	    #sR_TRIG_FlowSplitterDownTime(CLK := #sx_AutomaticActive AND NOT #sx_Ready);     // Rising edge conveyor conveyor down

	    #sR_TRIG_AirPressureError(CLK := NOT #ix_AirPressureOk);                         // Rising edge air pressure error

	    #sR_TRIG_DebrisDetected(CLK := #ix_DebrisSensor);                                // Rising edge debris detection

	    #sR_TRIG_EnconderError(CLK := #ix_FlowSplitterEncoderError);                    // Rising edge encoder error

	    #sR_TRIG_Mode1(CLK := (#si_Mode = 1));                                          // Rising edge Mode 1

	    #sR_TRIG_Mode2(CLK := (#si_Mode = 2));                                          // Rising edge Mode 2

	    #sR_TRIG_Mode3(CLK := (#si_Mode = 3));                                          // Rising edge Mode 3

	    #sR_TRIG_Mode4(CLK := (#si_Mode = 4));                                          // Rising edge Mode 4

	    #sR_TRIG_Mode5(CLK := (#si_Mode = 5));                                          // Rising edge Mode 5

	    #sR_TRIG_EnergySave(CLK := #sUDT_CommonStatus.EnergySave);                     // Rising edge trigger Energy save mode.

	    // Timers

	    #PEC_TimerOnOffDelay(iudi_OnDelayTime := #iUDT_FlowSplitterConfiguration.PEC_EoSTimeOnDelay,                       // Off delay time to filter PEC signal
	                         iudi_OffDelayTime := #iUDT_FlowSplitterConfiguration.PEC_EoSTimeOffDelay,                     // On delay time to filter PEC signal
	                         ix_SignalToDelay := #ix_PECEos,                                                               // PEC input signal
	                         ix_Enable := #iUDT_FlowSplitterConfiguration.PEC_Present,                                     // PEC present bit is true if the flow splitter is equiped with PEC
	                         qx_DelayedSignal => #sx_PEC_EoSFiltered);                                                      // PEC signal filtered

	    #PEC_ChuteTimerOnOffDelay(iudi_OnDelayTime := #iUDT_FlowSplitterConfiguration.PEC_FilterChuteTimeOnDelay,          // Off delay time to filter chute PEC signal
	                              iudi_OffDelayTime := #iUDT_FlowSplitterConfiguration.PEC_FilterChuteTimeOffDelay,        // On delay time to filter chute PEC signal
	                              ix_SignalToDelay := #ix_PECDivertChute,                                                  // PEC chute signal
	                              ix_Enable := TRUE,                                                                        // Enable function
	                              qx_DelayedSignal => #sx_PEC_ChuteFiltered);                                               // PEC chute siganl filtered

	    #PEC_UpstreamTimerOnOffDelay(iudi_OnDelayTime := #iUDT_FlowSplitterConfiguration.PEC_FilterUpstreamTimeOnDelay,    // On delay time to filter upstream PEC
	                                 iudi_OffDelayTime := #iUDT_FlowSplitterConfiguration.PEC_FilterUpstreamTimeOffDelay,  // Off delay time to filter upstream PEC
	                                 ix_SignalToDelay := #ix_PECUpstream,                                                  // Signal to filter upstream PEC
	                                 ix_Enable := TRUE,                                                                     // Function enable
	                                 qx_DelayedSignal => #sx_PEC_UpstreamFiltered);                                         // Upstream PEC signal filtered

	    #sFB_DivertsActivationTimer(iudi_OnDelayTime := 0,
	                                iudi_OffDelayTime := #iUDT_FlowSplitterConfiguration.DivertsTimeActivation,                // Off delay to pop-up diverts
	                                ix_SignalToDelay := NOT #sx_PEC_UpstreamFiltered,                                           // Upstream signal filtered,
	                                ix_Enable := TRUE,
	                                qx_DelayedSignal => #sx_EnableDiverts);                                                     // Enabling diverts pop-up

	END_REGION

	REGION 2 - Reset faults

	    // Send reset request TO interface UDT
	    #iqUDT_FlowSplitterInterface.InternalErrorReset := #iqUDT_EquipmentControl.Command.Reset;
	    #iqUDT_FlowSplitterInterface.ResetStatistics := #iqUDT_EquipmentControl.Command.ResetData;

	    // Reset errors
	    // Reset PEC Jam if PEC is clear and reset command is received.
	    IF #iqUDT_EquipmentControl.Command.Reset THEN                      // Reset bit from control block

	        IF #ix_PECEos = TRUE THEN
	            #sUDT_HMIStatus.Specific.PEC_EoSJam := FALSE;                     // PEC jam reset
	        END_IF;

	        IF #ix_DebrisSensor = TRUE THEN
	            #sUDT_HMIStatus.Specific.Debris := FALSE;                         // Debris fault reset
	        END_IF;

	        IF #ix_PECDivertChute = TRUE THEN
	            #sUDT_HMIStatus.Specific.PEC_DivertChuteJam := FALSE;             // Divert chute jam reset
	        END_IF;

	        IF #ix_AirPressureOk = TRUE THEN
	            #sUDT_HMIStatus.Specific.AirPressure := FALSE;                    // Air pressure error reset
	        END_IF;

	        IF #ix_FlowSplitterEncoderError = FALSE THEN
	            #sUDT_HMIStatus.Specific.EncoderError := FALSE;                   // Encoder error reset
	        END_IF;

	    END_IF;

	    // Error
	    #sUDT_CommonStatus.Error := NOT #ix_SafetyOk                               // safety error status
	    OR #sUDT_HMIStatus.Specific.EncoderError                                   // Enconder error status
	    OR #sUDT_HMIStatus.Specific.PEC_EoSJam                                     // PEC blockage error status
	    OR #sUDT_HMIStatus.Specific.PEC_DivertChuteJam                             // PEC divert chute blockage error status
	    OR #sUDT_HMIStatus.Specific.Debris                                         // Debris detected error status
	    OR #sUDT_HMIStatus.Specific.DivertsActivationError                         // Diverts position error status
	    OR #iqUDT_FlowSplitterInterface.InternalErrorVFD                           // Internal VFD error status
	    OR NOT #ix_Connected                                                        // Isolator switch error status
	    OR #iqUDT_FlowSplitterInterface.InternalErrorPEC;                          // External PEC fault
	    // Warning
	    #sUDT_CommonStatus.Warning := #sUDT_HMIStatus.Specific.AirPressure;       // Air pressure status;

	    // Ready
	    #sx_Ready := NOT #sUDT_CommonStatus.Error                                  // Ready bit is set true when common error status its false
	    AND #ix_24vOk                                                               // 24V is okay
	    AND #ix_400vOk                                                              // 400V is okay
	    AND NOT #iqUDT_FlowSplitterInterface.ConfigurationError;                   // not configuration error

	END_REGION

	REGION 3 - Stop conveyor

	    // Conditions to stop conveyor
	    IF ((#sF_TRIG_RunManual.Q OR #sF_TRIG_Jog.Q) AND #sx_ManualModeActive)                        // If in manula mode and Rising or falling edge for jog occur
	        OR (NOT #iqUDT_EquipmentControl.Command.AutomaticOn AND NOT #sx_ManualModeActive)      // or Not automatic ON and Not in manual mode
	        OR (NOT #sx_Ready AND NOT #sx_ManualModeActive)                                         // Or not ready and not in automatic mode
	        OR (#sR_TRIG_ManualMode.Q OR #sF_TRIG_ManualMode.Q)                                       // or Rising edge or falling edge of manual mode active command occur
	        OR NOT #ix_SafetyOk                                                                     // or safety not ok

	    THEN
	        //  Order to stop VFD
	        #iqUDT_FlowSplitterInterface.RunFwd := FALSE;                  // Reset order to VFD run in forward direction
	        #iqUDT_FlowSplitterInterface.RunRvs := FALSE;                  // Reset order to VFD run in reverse direction
	        #iqUDT_HandShakeUp.RTR := FALSE;                               // Reset the bit ready to receive
	        #iqUDT_HandShakeUp.CascadeStartUp := FALSE;                    // Reset cascade start up bit

	        #sx_AutomaticActive := FALSE;                                   // Automatic mode is disable
	        #sx_StartReceived := FALSE;                                     // Clear start receive bit

	        #sx_Zone1_Divert := FALSE;                                      // Reset diverts from zone 1
	        #sx_Zone2_Divert := FALSE;                                      // Reset diverts from zone 2

	        #sx_Switch1To3 := FALSE;                                        // Reset switch from mode 1 to mode 3 auxiliary bit
	        #sx_Switch3To1 := FALSE;                                        // Reset switch from mode 3 to mode 1 auxiliary bit
	    END_IF;

	END_REGION

	REGION 4 - Start
	    // Save Start bit request
	    IF NOT #sx_ManualModeActive                                         // If Manual mode iis not active
	        AND #sx_Ready                                                   // and Flow splitter is ready
	        AND #iqUDT_EquipmentControl.Command.Start                      // Start command from control block received
	        AND #iqUDT_EquipmentControl.Command.AutomaticOn                // Automatic on signal from control block is active
	    THEN                                                                // then
	        #sx_StartReceived := TRUE;                                      // Set start received bit
	    END_IF;

	    // Cascade mode

	    CASE #si_Mode OF
	        1:  // Statement section case 1 (Flow splitter in straight direction)
	            IF #sx_StartReceived                                                 // If Start received memory bit is active
	                AND (#iqUDT_HandShakeStraight.CascadeStartUp                    // And Cascade start bit from downstream straight conveyor handshake is active
	                OR #iUDT_FlowSplitterConfiguration.FirstConveyorToStart)        // Or flow splitter conveyor is the first conveyor to start
	            THEN                                                                 // then
	                #sx_AutomaticActive := TRUE;                                     // Automatic active is set true
	                #sx_StartReceived := FALSE;                                      // and reset start received memory bit
	            END_IF;
	            ;
	        3:  // Statement section case 3 (Flow splitter in divert direction)
	            IF #sx_StartReceived                                                 // If Start received memory bit is active
	                AND (#iqUDT_HandShakeDivert.CascadeStartUp                      // And Cascade start bit from downstream divert conveyor handshake is avtive
	                OR #iUDT_FlowSplitterConfiguration.FirstConveyorToStart)        // Or flow splitter conveyor is the first conveyor to start
	            THEN                                                                 // Then
	                #sx_AutomaticActive := TRUE;                                     //  Automatic active is set true
	                #sx_StartReceived := FALSE;                                      //and reset start received memory bit
	            END_IF;
	            ;
	        ELSE  // Statement section ELSE
	            IF #sx_StartReceived                                                 // If Start received memory bit is activ
	                AND (#iqUDT_HandShakeStraight.CascadeStartUp                    // And Cascade start bit from downstream straight conveyor handshake is active
	                AND #iqUDT_HandShakeDivert.CascadeStartUp                       // And Cascade start bit from downstream divert conveyor handshake is active
	                OR #iUDT_FlowSplitterConfiguration.FirstConveyorToStart)        // Or flow splitter conveyor is the first conveyor to start
	            THEN                                                                 // Then
	                #sx_AutomaticActive := TRUE;                                     // Automatic active is set true
	                #sx_StartReceived := FALSE;                                      // and reset start received memory bit
	            END_IF;
	            ;
	    END_CASE;

	    //Timer to cascade mode

	    #sFB_CascadeModeTimer(iudi_OnDelayTime := #iUDT_FlowSplitterConfiguration.CascadeTimeOnDelay,      // Cascade mode timer
	                          ix_SignalToDelay := #sx_AutomaticActive,                                      // Signal to activate the timer
	                          ix_Enable := #sx_Ready,                                                       // Bit ready to enable cascade mode
	                          qx_DelayedSignal => #iqUDT_HandShakeUp.CascadeStartUp);                      // Cascade mode signal to upstream

	END_REGION

	REGION 5 - Manual mode

	    // Manual mode activation
	    #sx_ManualModeActive := #iqUDT_FlowSplitterCommand.ManualMode                                  // Manual mode is active if the bits that activate manual mode is active from hmi or from control block
	    OR #iqUDT_EquipmentControl.Command.ManualMode;

	    //Send manual mode active to PEC/VFD blocks to supress errors
	    #iqUDT_FlowSplitterInterface.ManualModeActive := #sx_ManualModeActive;

	    //When the system is not any more in manual mode or when fatal error occurs the HMI commands should be reset

	    IF NOT #ix_SafetyOk
	        OR NOT #ix_24vOk                                                        // 24V error status
	        OR NOT #ix_400vOk                                                       // 400V error status
	        OR NOT #ix_HardwareOk                                                   // Profinet error status
	        OR #iqUDT_FlowSplitterInterface.ConfigurationError                          // No configuration err
	        OR #iqUDT_FlowSplitterInterface.InternalErrorVFD
	        OR #iqUDT_FlowSplitterInterface.Disconnected
	        OR NOT #sx_ManualModeActive
	    THEN
	        #iqUDT_FlowSplitterCommand.ManualStartStop := FALSE;
	        #iqUDT_FlowSplitterCommand.ManualFullSpeed := FALSE;
	        #iqUDT_FlowSplitterCommand.ManualJog := FALSE;
	    END_IF;

	    // Manual mode force disable
	    IF #iqUDT_EquipmentControl.Command.DisableManualMode THEN
	        #iqUDT_FlowSplitterCommand.ManualMode := False;
	        #iqUDT_FlowSplitterCommand.ManualFullSpeed := False;
	        #iqUDT_FlowSplitterCommand.ManualJog := False;
	        #iqUDT_FlowSplitterCommand.ManualStartStop := False;
	    END_IF;

	    // Start/Stop in manual mode
	    IF #sx_ManualModeActive THEN                                            // If Manual mode is active then check prestart status for manual mode
	        #sx_PreStartManual := #ix_SafetyOk                                  // If Safety is Okay
	        AND #ix_Connected                                                   // And Isolator switch is connected
	        AND #ix_HardwareOk                                                  // And Profinet connection is okay
	        AND NOT #iqUDT_FlowSplitterInterface.InternalErrorVFD;             // Add no error on VFD // Then conveyor is allowed to run in manual mode.

	        IF (#sx_PreStartManual                                                              // If Pre start conditions to run in manual mode is okay
	            AND (#sR_TRIG_RunManual.Q AND NOT #iqUDT_FlowSplitterCommand.ManualJog)         // and rising edge to run in manual mode is detected and it is not running in jogging mode
	            OR (#sR_TRIG_Jog.Q AND NOT #iqUDT_FlowSplitterCommand.ManualStartStop))         // Or rising edge to start jogging is detected and it is not running in manual mode
	        THEN
	            #iqUDT_EquipmentControl.Request.SignalingRequest := TRUE;                      //then Request signaling to control block before conveyor run in manual mode
	        END_IF;

	        // To Run conveyor forward in manual mode
	        #iqUDT_FlowSplitterInterface.RunFwd := #sx_PreStartManual          // Prestart conditions to run in manual mode is active
	        AND NOT #iqUDT_EquipmentControl.Request.SignalingRequest           // And Signaling request done
	        AND (#iqUDT_FlowSplitterCommand.ManualStartStop                    // And Command to manual Run or manual jog is active
	        OR #iqUDT_FlowSplitterCommand.ManualJog);                          // Then run motor in forward direction

	        // Flow splitter belt should not run in reverse direction
	        #iqUDT_FlowSplitterInterface.RunRvs := FALSE;

	        // Pop up diverts in manual mode
	        #sx_Zone1_Divert := #sx_PreStartManual AND #iqUDT_FlowSplitterCommand.Zone1DivertActivation;          // Output bit to active zone 1 diverts
	        #sx_Zone2_Divert := #sx_PreStartManual AND #iqUDT_FlowSplitterCommand.Zone2DivertActivation;          // Output bit to active zone 2 diverts

	    END_IF;

	END_REGION

	REGION 6 - Automatic mode active

	    IF NOT #sx_ManualModeActive THEN                                        // Manual mode is not active
	        IF #sx_AutomaticActive AND #sx_Ready THEN                           // Automatic mode active AND ready

	            #iqUDT_HandShakeUp.RTR := #iqUDT_FlowSplitterInterface.VFDatSpeed;            // Ready to receive handshake to upstream if VFD is at speed

	            CASE #si_Mode OF                                                // Operation mode case selection

	                1:  // 100% straight

	                    // Order to VFD to run
	                    #iqUDT_FlowSplitterInterface.RunFwd := NOT #ix_ExternalRequestHold             // Halt request is not active
	                    AND #iqUDT_HandShakeStraight.RTR                                               // Ready to receive active
	                    AND NOT #sx_EnergySaveActive;                                                   // Energy save is not active

	                    #sx_Zone2_Divert := FALSE;                                                      // Output bit to active zone 2 diverts
	                    #sx_Zone1_Divert := #sx_Switch3To1;                                             // Output bit to active zone 1 diverts

	                    IF #sx_Switch3To1 THEN                                                          // Memory bit switch from mode 3 to mode 1
	                        IF "DB_Memory".OS_1sec THEN                                                 // Memory bit 1 second trigger
	                            #si_SwitchDelay += 1;                                                   // Memory integer to count time to delay switch
	                        END_IF;

	                        IF #si_SwitchDelay >= #iUDT_FlowSplitterConfiguration.DivertSwitchDelay THEN    // Comparation between memory integer switch delay and configuration divert switch delay
	                            #si_SwitchDelay := 0;                                                   // Reset memory integer switch delay counter
	                            #sx_Switch3To1 := FALSE;                                                // Reset switch from mode 3 to mode 1 memory bit
	                        END_IF;
	                    END_IF;

	                    #sx_Switch1To3 := TRUE;                                                         // Set memory bit switch from mode 1 to mode 3
	                    ;

	                2:  // 50% straight - 50% divert

	                    #iqUDT_FlowSplitterInterface.RunFwd := ((#iqUDT_HandShakeStraight.RTR         // Ready to receive downstream straight
	                    AND #iqUDT_HandShakeDivert.RTR)                                                // Ready to receive downstream divert chute
	                    OR (#iUDT_FlowSplitterConfiguration.OnFlyChangeOfMode                          // On fly change mode
	                    AND (#iqUDT_HandShakeStraight.RTR                                              // Ready to receive downstream straight
	                    OR (#iqUDT_HandShakeDivert.RTR AND NOT #sUDT_HMIStatus.Specific.AirPressure))))// Ready to receive downstream divert chute
	                    //   AND (NOT #i_UDT_FlowSplitterConfiguration.OnFlyChangeOfMode
	                    //   AND NOT #s_UDT_HMIStatus.Specific.AirPressure)
	                    AND NOT #ix_ExternalRequestHold                                                // External requesto to halt
	                    AND NOT #sx_EnergySaveActive;                                                   // Energy save is not active

	                    #sx_Zone1_Divert := (#iqUDT_HandShakeDivert.RTR                                // Ready to receive downstream divert chute
	                    OR NOT #iqUDT_HandShakeStraight.RTR                                            // Ready to receive downstream straight
	                    OR NOT #iUDT_FlowSplitterConfiguration.OnFlyChangeOfMode)                      // On fly change mode
	                    AND NOT #sUDT_HMIStatus.Specific.AirPressure;                                         // And Air pressure is OK

	                    #sx_Zone2_Divert := (#iUDT_FlowSplitterConfiguration.OnFlyChangeOfMode         // On fly change mode
	                    AND NOT #iqUDT_HandShakeStraight.RTR                                           // Ready to receive downstream straight
	                    AND #iqUDT_HandShakeDivert.RTR)
	                    AND NOT #sUDT_HMIStatus.Specific.AirPressure;                                         // Ready to receive downstream divert chute

	                    #sx_Switch1To3 := FALSE;                                                        // Switch from mode 1 to mode 3
	                    #sx_Switch3To1 := FALSE;                                                        // Switch from mode 3 to mode 1
	                    ;

	                3:  // 0% straight - 100% divert

	                    // Order to VFD to run
	                    #iqUDT_FlowSplitterInterface.RunFwd := NOT #ix_ExternalRequestHold             // Halt request is not active
	                    AND #iqUDT_HandShakeDivert.RTR                                                 // Handshake Ready to receive from downstream divert conveyor
	                    AND NOT #sUDT_HMIStatus.Specific.AirPressure
	                    AND NOT #sx_EnergySaveActive;                                                   // Energy save is not active

	                    #sx_Zone1_Divert := NOT #sUDT_HMIStatus.Specific.AirPressure;                         // Output bit to active zone 1 diverts
	                    #sx_Zone2_Divert := NOT #sx_Switch1To3 AND NOT #sUDT_HMIStatus.Specific.AirPressure;  // Output bit to active zone 2 diverts

	                    IF #sx_Switch1To3 THEN                                                          // Memory bit switch mode 1 to mode 3
	                        IF "DB_Memory".OS_1sec THEN                                                 // Memory bit 1 second trigger
	                            #si_SwitchDelay += 1;                                                   // Memory integer to count time to delay switch
	                        END_IF;

	                        IF #si_SwitchDelay > #iUDT_FlowSplitterConfiguration.DivertSwitchDelay     // Comparation between memory integer switch delay and configuration divert switch delay
	                        THEN
	                            #si_SwitchDelay := 0;                                                   // Reset memory integer switch delay counter
	                            #sx_Switch1To3 := FALSE;                                                // Reset switch from mode 1 to mode 3 memory bit
	                        END_IF;
	                    END_IF;
	                    #sx_Switch3To1 := TRUE;                                                         // Set memory bit switch from mode 3 to mode 1
	                    ;

	                4:  // Based on time

	                    #iqUDT_FlowSplitterInterface.RunFwd := ((#iqUDT_HandShakeStraight.RTR         // Ready to receive downstream straight
	                    AND #iqUDT_HandShakeDivert.RTR)                                                // Ready to receive downstream divert chute
	                    OR (#iUDT_FlowSplitterConfiguration.OnFlyChangeOfMode                          // On fly change mode
	                    AND (#iqUDT_HandShakeStraight.RTR                                              // Ready to receive downstream straight
	                    OR (#iqUDT_HandShakeDivert.RTR AND NOT #sUDT_HMIStatus.Specific.AirPressure))))      // Ready to receive downstream divert chute
	                    //  AND (NOT #i_UDT_FlowSplitterConfiguration.OnFlyChangeOfMode
	                    //  AND NOT #s_UDT_HMIStatus.Specific.AirPressure)
	                    AND NOT #ix_ExternalRequestHold                                                 // External requesto to halt
	                    AND NOT #sx_EnergySaveActive;                                                   // Energy save is not active

	                    #sx_Switch1To3 := FALSE;                                                        // Reset switch from mode 1 to mode 3 memory bit
	                    #sx_Switch3To1 := FALSE;                                                        // Reset switch from mode 3 to mode 1 memory bit

	                    #si_Mode4DivertTime := REAL_TO_INT(#iqUDT_FlowSplitterCommand.PercentageSplit * #iUDT_FlowSplitterConfiguration.TimeBasedSplit) / 100;      // Memory integer to calculate time base

	                    IF "DB_Memory".OS_1sec AND #iqUDT_HandShakeDivert.RTR THEN                     // Memory bit 1 second trigger and Handshake bit ready to receive to upstream
	                        #si_Mode4AuxTimer += 1;                                                     // Increment counter to time base mode
	                    END_IF;

	                    #tx_AuxBaseTimeDivert1 := FALSE;                                                // Auxiliary base time divert zone 1
	                    #tx_AuxBaseTimeDivert2 := FALSE;                                                // Auxiliary base time divert zone 2

	                    IF (#si_Mode4AuxTimer <= #si_Mode4DivertTime)                                   // If the counter time is lower than calculated time from configuration
	                    THEN
	                        #tx_AuxBaseTimeDivert1 := TRUE;                                             // Auxiliary base time divert zone 1
	                        #tx_AuxBaseTimeDivert2 := TRUE;                                             // Auxiliary base time divert zone 2
	                    END_IF;

	                    IF (#si_Mode4AuxTimer > #si_Mode4DivertTime)                                    // If the counter time is bigger than calculated time from configuration
	                        AND (#si_Mode4AuxTimer < #iUDT_FlowSplitterConfiguration.TimeBasedSplit)   // If the counter time is lower than time based split configured
	                    THEN
	                        #tx_AuxBaseTimeDivert1 := FALSE;                                            // Auxiliary base time divert zone 1
	                        #tx_AuxBaseTimeDivert2 := FALSE;                                            // Auxiliary base time divert zone 2
	                    END_IF;

	                    IF (#si_Mode4AuxTimer >= #iUDT_FlowSplitterConfiguration.TimeBasedSplit) THEN  // If the counter time is bigger or equal than time based split configured
	                        #si_Mode4AuxTimer := 0;                                                     // Reset counter time
	                    END_IF;

	                    IF (#iqUDT_HandShakeDivert.RTR                                                 // Ready to receive downstream divert chute
	                        AND ((#tx_AuxBaseTimeDivert1 AND #tx_AuxBaseTimeDivert2)
	                        OR (NOT #iqUDT_HandShakeStraight.RTR AND #iUDT_FlowSplitterConfiguration.OnFlyChangeOfMode)))
	                        AND NOT #sUDT_HMIStatus.Specific.AirPressure
	                    THEN
	                        #sx_Zone1_Divert := TRUE;
	                        #sx_Zone2_Divert := TRUE;

	                    ELSIF #iqUDT_HandShakeStraight.RTR
	                        AND ((NOT #tx_AuxBaseTimeDivert1 AND NOT #tx_AuxBaseTimeDivert2)
	                        OR (NOT #iqUDT_HandShakeDivert.RTR AND #iUDT_FlowSplitterConfiguration.OnFlyChangeOfMode))
	                        OR #sUDT_HMIStatus.Specific.AirPressure
	                    THEN
	                        #sx_Zone1_Divert := FALSE;
	                        #sx_Zone2_Divert := FALSE;
	                    END_IF
	                    ;

	                5:  // Semi automatic mode

	                    #iqUDT_FlowSplitterInterface.RunFwd := NOT #ix_ExternalRequestHold     // External requesto to halt
	                    AND NOT #sx_EnergySaveActive                                            // Energy save is not active
	                    AND ((#iqUDT_HandShakeStraight.RTR                                     // Ready to receive downstream straight
	                    AND NOT #iqUDT_FlowSplitterCommand.Zone1DivertActivation               // Command divert activation zone 1
	                    AND NOT #iqUDT_FlowSplitterCommand.Zone2DivertActivation)              // Command divert activation zone 2
	                    OR (#iqUDT_HandShakeDivert.RTR                                         // Ready to receive downstream divert chute
	                    AND #iqUDT_FlowSplitterCommand.Zone1DivertActivation                   // Command divert activation zone 1
	                    AND #iqUDT_FlowSplitterCommand.Zone2DivertActivation                   // Command divert activation zone 2
	                    AND NOT #sUDT_HMIStatus.Specific.AirPressure)                                 // Air preassure is OK
	                    OR (#iqUDT_HandShakeStraight.RTR                                       // Ready to receive downstream straight
	                    AND #iqUDT_HandShakeDivert.RTR                                         // Ready to receive downstream divert chute
	                    AND #iqUDT_FlowSplitterCommand.Zone1DivertActivation                   // Command divert activation zone 1
	                    AND NOT #iqUDT_FlowSplitterCommand.Zone2DivertActivation               // Command divert activation zone 2
	                    AND NOT #sUDT_HMIStatus.Specific.AirPressure));

	                    #sx_Zone1_Divert := #iqUDT_FlowSplitterCommand.Zone1DivertActivation   // Command divert activation zone 1
	                    AND NOT #sUDT_HMIStatus.Specific.AirPressure;

	                    #sx_Zone2_Divert := #iqUDT_FlowSplitterCommand.Zone2DivertActivation   // Command divert activation zone 2
	                    AND NOT #sUDT_HMIStatus.Specific.AirPressure;

	                    #sx_Switch1To3 := FALSE;                                                // Reset switch from mode 1 to mode 3 memory bit
	                    #sx_Switch3To1 := FALSE;                                                // Reset switch from mode 3 to mode 1 memory bit
	                    ;
	            END_CASE;

	            // Flow splitter end OF section PEC jam

	            IF #iUDT_FlowSplitterConfiguration.PEC_Present THEN

	                IF NOT #sx_PEC_EoSFiltered AND #ix_HardwareOk THEN                                      // Photo eye blocked
	                    #si_AuxJamDisplacement += #iqUDT_FlowSplitterInterface.Displacement;               // Increases displacement values in auxiliary variable
	                ELSE
	                    #si_AuxJamDisplacement := 0;                                                        // Reset jam auxiliary counter variable
	                END_IF;

	                IF #si_AuxJamDisplacement > #iUDT_FlowSplitterConfiguration.JamDisplacementLimit THEN  // Compare jam auxiliary counter with displacement jam configured
	                    #sUDT_HMIStatus.Specific.PEC_EoSJam := TRUE;                                              // PEC jam status set true
	                END_IF;

	            END_IF;

	            // Chute PEC jam

	            IF #iUDT_FlowSplitterConfiguration.PEC_ChutePesent THEN
	                IF NOT #sx_PEC_ChuteFiltered AND #ix_HardwareOk THEN
	                    #si_AuxJamDivertChuteDisplacement += #iqUDT_FlowSplitterInterface.Displacement;
	                ELSE
	                    #si_AuxJamDivertChuteDisplacement := 0;
	                END_IF;

	                IF #si_AuxJamDivertChuteDisplacement > #iUDT_FlowSplitterConfiguration.DivertChuteJamDisplacLimit THEN     // Compare jam auxiliary counter with displacement jam configured
	                    #sUDT_HMIStatus.Specific.PEC_DivertChuteJam := TRUE;                                                          // PEC jam status set true
	                END_IF;

	            END_IF;

	            // Debris detection
	            #sFB_DebrisTimer(iudi_OnDelayTime := #iUDT_FlowSplitterConfiguration.DebrisTimeFilter,      // Debris filtering time configuration
	                             iudi_OffDelayTime := 0,
	                             ix_SignalToDelay := NOT #ix_DebrisSensor AND #ix_HardwareOk,                // Debris sensor signal input
	                             ix_Enable := TRUE,                                                          // Enable timer
	                             qx_DelayedSignal => #sx_DebrisSignalFiltered);                              // Debris sensor signal filtered

	            #sUDT_HMIStatus.Specific.Debris := #sx_DebrisSignalFiltered;                                              // Debris error status

	            // Energy save
	            #iqUDT_HandShakeStraight.ResetEnergySave := NOT #ix_PECUpstream;
	            #iqUDT_HandShakeDivert.ResetEnergySave := NOT #ix_PECUpstream AND #sx_EnableDiverts;

	        ELSE
	            // If conveyor is not in manual mode and not ready
	            #iqUDT_FlowSplitterInterface.RunFwd := FALSE;                                                      // Order to VFD stop conveyor
	            #iqUDT_HandShakeUp.RTR := FALSE;                                                                   // Set ready to receive false

	        END_IF;
	    END_IF;

	    // Air pressure error
	    IF NOT #ix_AirPressureOk AND #ix_HardwareOk THEN
	        #sUDT_HMIStatus.Specific.AirPressure := TRUE;
	    END_IF;

	    // Encoder error
	    IF #ix_FlowSplitterEncoderError AND #ix_HardwareOk THEN
	        #sUDT_HMIStatus.Specific.EncoderError := TRUE;
	    END_IF;

	    // Diverts output control
	    #qx_Zone1Divert := #sx_Zone1_Divert AND (#sx_EnableDiverts OR NOT #iUDT_FlowSplitterConfiguration.DivertsTimeSave);
	    #qx_Zone2Divert := #sx_Zone2_Divert AND (#sx_EnableDiverts OR NOT #iUDT_FlowSplitterConfiguration.DivertsTimeSave);

	    // Divert activation error is true when the diverts from zone 2 is active and the diverts from zone 1 is not pop up.
	    #sUDT_HMIStatus.Specific.DivertsActivationError := NOT #qx_Zone1Divert AND #qx_Zone2Divert;

	    // Update mode status for HMI, IF not in manual mode update selected mode otherwise write 0
	    IF NOT #sx_ManualModeActive THEN
	        #sUDT_HMIStatus.Specific.Mode := #si_Mode;
	    ELSE
	        #sUDT_HMIStatus.Specific.Mode := 0;
	    END_IF;

	    //Update actual direction status of divert for HMI
	    #sUDT_HMIStatus.Specific.Zone1Divert := #qx_Zone1Divert;
	    #sUDT_HMIStatus.Specific.Zone2Divert := #qx_Zone2Divert;

	END_REGION

	REGION 7 - Energy save

	    IF #iUDT_FlowSplitterConfiguration.Energy THEN

	        // Set Energy save active.
	        IF #si_AuxEnergySave >= #iUDT_FlowSplitterConfiguration.EnergySaveLength
	        THEN
	            #sx_EnergySaveActive := TRUE;
	        END_IF;

	        IF ((NOT #sx_PEC_EoSFiltered AND #iUDT_FlowSplitterConfiguration.PEC_Present)
	            OR #iqUDT_HandShakeUp.RTS
	            OR #iqUDT_HandShakeUp.ResetEnergySave
	            OR #ix_ResetEnergySave
	            OR #sx_ManualModeActive)
	        THEN
	            #si_AuxEnergySave := 0;
	            #sx_EnergySaveActive := FALSE;
	        ELSE
	            #si_AuxEnergySave += #iqUDT_FlowSplitterInterface.Displacement;
	        END_IF;

	    ELSE

	        #si_AuxEnergySave := 0;
	        #sx_EnergySaveActive := FALSE;

	    END_IF;



	END_REGION

	REGION 8 - Speed control
	    (*In manual mode, conveyor runs with low speed by default. If "ManualFullSpeed" is set true, conveyor runs with high speed in manual mode.
	      In automatic mode, conveyor runs with full speed if external is zero. If external speed is bigger than zero, conveyor will run with that speed. *)

	    IF #sx_ManualModeActive                                                                                 // Manual mode active
	    THEN
	        IF #iqUDT_FlowSplitterCommand.ManualFullSpeed                                                      // Full speed in manual mode
	            AND #iqUDT_FlowSplitterCommand.ManualStartStop                                                 // Start/stop conveyor in manual mode
	        THEN
	            #iqUDT_FlowSplitterInterface.SpeedSetpoint := #iUDT_FlowSplitterConfiguration.SpeedSetpointNominal;   // Move nominal setpoint to the VDF
	        ELSE
	            #iqUDT_FlowSplitterInterface.SpeedSetpoint := #iUDT_FlowSplitterConfiguration.SpeedSetpointLow;       // Move low speed setpoint to VFD
	        END_IF;

	    ELSE

	        IF #iui_ExternalSpeed > 0                                                                           // If external speed bigger than zero
	        THEN
	            #iqUDT_FlowSplitterInterface.SpeedSetpoint := #iui_ExternalSpeed;                                      // Move external speed to VFD
	        ELSE
	            #iqUDT_FlowSplitterInterface.SpeedSetpoint := #iUDT_FlowSplitterConfiguration.SpeedSetpointNominal;   // Move nominal setpoint to VFD
	        END_IF;

	    END_IF;

	END_REGION

	REGION 9 - Statistics

	    // Flow splitter up Time
	    IF #sx_AutomaticActive AND #sx_Ready OR #iqUDT_EquipmentControl.Command.ResetData THEN                 // Automatic active
	        "FC_Statistics"(ix_Reset := #iqUDT_EquipmentControl.Command.ResetData,                             // Reset statistics input
	                        ix_Activate := #sx_AutomaticActive                                                  // Activate statistics functions input
	                        AND #sx_Ready,
	                        ix_RTrigActivate := #sR_TRIG_FlowSplitterUpTime.Q,                                   // Statistics active trigger
	                        iqUDT_Statistics := #iqUDT_Statistics.FlowSplitterUpTime);                        // Statistics values output
	    END_IF;

	    // 9.2 - Flow splitter down Time
	    IF #sx_AutomaticActive AND NOT #sx_Ready OR #iqUDT_EquipmentControl.Command.ResetData THEN             // Automatic active
	        "FC_Statistics"(ix_Reset := #iqUDT_EquipmentControl.Command.ResetData,                             // Reset statistics input
	                        ix_Activate := #sx_AutomaticActive                                                  // Activate statistics functions input
	                        AND NOT #sx_Ready,
	                        ix_RTrigActivate := #sR_TRIG_FlowSplitterDownTime.Q,                                 // Statistics active trigger
	                        iqUDT_Statistics := #iqUDT_Statistics.FlowSplitterDownTime);                      // Statistics values output
	    END_IF;

	    // Chute PEC Blockage error
	    IF #sUDT_HMIStatus.Specific.PEC_DivertChuteJam OR #iqUDT_EquipmentControl.Command.ResetData THEN             // PEC jam error active
	        "FC_Statistics"(ix_Reset := #iqUDT_EquipmentControl.Command.ResetData,                             // Reset statistics input
	                        ix_Activate := #sUDT_HMIStatus.Specific.PEC_DivertChuteJam,                               // Activate statistics functions input
	                        ix_RTrigActivate := #sR_TRIG_PECDivertChuteJam.Q,                                    // Statistics active trigger
	                        iqUDT_Statistics := #iqUDT_Statistics.PECChuteDivertJam);                         // Statistics values output
	    END_IF;

	    // PEC Blockage error
	    IF (#sUDT_HMIStatus.Specific.PEC_EoSJam OR #iqUDT_EquipmentControl.Command.ResetData) THEN                   // PEC jam error active
	        "FC_Statistics"(ix_Reset := #iqUDT_EquipmentControl.Command.ResetData,                             // Reset statistics input
	                        ix_Activate := #sUDT_HMIStatus.Specific.PEC_EoSJam,                                       // Activate statistics functions input
	                        ix_RTrigActivate := #sR_TRIG_PECJam.Q,                                               // Statistics active trigger
	                        iqUDT_Statistics := #iqUDT_Statistics.PEC_EoSJam);                                // Statistics values output
	    END_IF;

	    // Air pressure error
	    IF #sUDT_HMIStatus.Specific.AirPressure OR #iqUDT_EquipmentControl.Command.ResetData THEN
	        "FC_Statistics"(ix_Reset := #iqUDT_EquipmentControl.Command.ResetData,
	                        ix_Activate := #sUDT_HMIStatus.Specific.AirPressure,
	                        ix_RTrigActivate := #sR_TRIG_AirPressureError.Q,
	                        iqUDT_Statistics := #iqUDT_Statistics.AirPressure);
	    END_IF;

	    // Debris detecting
	    IF #sUDT_HMIStatus.Specific.Debris OR #iqUDT_EquipmentControl.Command.ResetData THEN
	        "FC_Statistics"(ix_Reset := #iqUDT_EquipmentControl.Command.ResetData,
	                        ix_Activate := #sUDT_HMIStatus.Specific.Debris,
	                        ix_RTrigActivate := #sR_TRIG_DebrisDetected.Q,
	                        iqUDT_Statistics := #iqUDT_Statistics.DebrisSensor);
	    END_IF;

	    // Encoder error
	    IF #ix_FlowSplitterEncoderError OR #iqUDT_EquipmentControl.Command.ResetData THEN
	        "FC_Statistics"(ix_Reset := #iqUDT_EquipmentControl.Command.ResetData,
	                        ix_Activate := #ix_FlowSplitterEncoderError,
	                        ix_RTrigActivate := #sR_TRIG_EnconderError.Q,
	                        iqUDT_Statistics := #iqUDT_Statistics.EncoderError);
	    END_IF;

	    // Mode 1
	    IF (#si_Mode = 1 AND NOT #sx_ManualModeActive) OR #iqUDT_EquipmentControl.Command.ResetData THEN
	        "FC_Statistics"(ix_Reset := #iqUDT_EquipmentControl.Command.ResetData,
	                        ix_Activate := (#si_Mode = 1)
	                        AND #iqUDT_FlowSplitterInterface.VFDRunning,
	                        ix_RTrigActivate := #sR_TRIG_Mode1.Q,
	                        iqUDT_Statistics := #iqUDT_Statistics.Mode100Divert);
	    END_IF;

	    // Mode 2
	    IF (#si_Mode = 2 AND NOT #sx_ManualModeActive) OR #iqUDT_EquipmentControl.Command.ResetData THEN
	        "FC_Statistics"(ix_Reset := #iqUDT_EquipmentControl.Command.ResetData,
	                        ix_Activate := (#si_Mode = 2)
	                        AND #iqUDT_FlowSplitterInterface.VFDRunning,
	                        ix_RTrigActivate := #sR_TRIG_Mode2.Q,
	                        iqUDT_Statistics := #iqUDT_Statistics."Mode50/50");
	    END_IF;

	    // Mode 3
	    IF (#si_Mode = 3 AND NOT #sx_ManualModeActive) OR #iqUDT_EquipmentControl.Command.ResetData THEN
	        "FC_Statistics"(ix_Reset := #iqUDT_EquipmentControl.Command.ResetData,
	                        ix_Activate := (#si_Mode = 3)
	                        AND #iqUDT_FlowSplitterInterface.VFDRunning,
	                        ix_RTrigActivate := #sR_TRIG_Mode3.Q,
	                        iqUDT_Statistics := #iqUDT_Statistics.Mode100Divert);
	    END_IF;

	    // Mode 4
	    IF (#si_Mode = 4 AND NOT #sx_ManualModeActive) OR #iqUDT_EquipmentControl.Command.ResetData THEN
	        "FC_Statistics"(ix_Reset := #iqUDT_EquipmentControl.Command.ResetData,
	                        ix_Activate := (#si_Mode = 4)
	                        AND #iqUDT_FlowSplitterInterface.VFDRunning,
	                        ix_RTrigActivate := #sR_TRIG_Mode4.Q,
	                        iqUDT_Statistics := #iqUDT_Statistics.ModeTimeBasedSplit);
	    END_IF;

	    // Mode 5
	    IF (#si_Mode = 5 AND NOT #sx_ManualModeActive) OR #iqUDT_EquipmentControl.Command.ResetData THEN
	        "FC_Statistics"(ix_Reset := #iqUDT_EquipmentControl.Command.ResetData,
	                        ix_Activate := (#si_Mode = 5)
	                        AND #iqUDT_FlowSplitterInterface.VFDRunning,
	                        ix_RTrigActivate := #sR_TRIG_Mode5.Q,
	                        iqUDT_Statistics := #iqUDT_Statistics.ModeSemiAutomatic);
	    END_IF;

	    // Enegry save mode
	    IF #sx_EnergySaveActive
	        OR #iqUDT_EquipmentControl.Command.ResetData
	    THEN
	        "FC_Statistics"(ix_Reset := #iqUDT_EquipmentControl.Command.ResetData,
	                        ix_Activate := #sUDT_CommonStatus.EnergySave,
	                        ix_RTrigActivate := #sR_TRIG_EnergySave.Q,
	                        iqUDT_Statistics := #iqUDT_Statistics.EnergySave);
	    END_IF;

	END_REGION

	REGION 10 - Status

	    #sUDT_CommonStatus.Stopped := #sx_Ready AND NOT #sx_AutomaticActive;               // stopped

	    #sUDT_CommonStatus.Running := #iqUDT_FlowSplitterInterface.RunFwd
	    OR #iqUDT_FlowSplitterInterface.RunRvs;                                            // Running

	    #sUDT_CommonStatus.Halted := #ix_ExternalRequestHold AND #sx_Ready AND #sx_AutomaticActive;   // Halted

	    #sUDT_CommonStatus.Dieback := #sx_Ready AND #sx_AutomaticActive
	    AND NOT #sUDT_CommonStatus.EnergySave
	    AND NOT #sUDT_CommonStatus.Running;                                                // Die back

	    #sUDT_CommonStatus.Manual := #sx_ManualModeActive;                                 // Manual

	    #sUDT_CommonStatus.ManualRun := #sx_ManualModeActive AND #sUDT_CommonStatus.Running;     // Manual Running

	    #sUDT_CommonStatus.EnergySave := #sx_EnergySaveActive;                             // Energy save active

	    #sUDT_CommonStatus.SafetyStop := NOT #ix_SafetyOk;                                 // Safety not ok

	    #sUDT_CommonStatus.Warning := #sUDT_HMIStatus.Specific.AirPressure;

	    IF #sUDT_CommonStatusOld <> #sUDT_CommonStatus THEN                               // update on change

	        // Set status to status number

	        #sUDT_HMIStatus.Status := 0;                                                   // Initialise status number

	        IF #sUDT_CommonStatus.EnergySave                                               // Energy save
	        THEN

	            #sUDT_HMIStatus.Status := "DB_HMIStatusConfiguration".EnergySave;

	        END_IF;

	        IF #sUDT_CommonStatus.Running                                                  // Running
	        THEN

	            #sUDT_HMIStatus.Status := "DB_HMIStatusConfiguration".Running;

	        END_IF;

	        IF #sUDT_CommonStatus.Stopped                                                  // Stopped
	        THEN

	            #sUDT_HMIStatus.Status := "DB_HMIStatusConfiguration".Stopped;

	        END_IF;

	        IF #sUDT_CommonStatus.Dieback                                                  // Dieback
	        THEN

	            #sUDT_HMIStatus.Status := "DB_HMIStatusConfiguration".Dieback;

	        END_IF;

	        IF #sUDT_CommonStatus.Halted                                                   // Halted
	        THEN

	            #sUDT_HMIStatus.Status := "DB_HMIStatusConfiguration".Halted;

	        END_IF;

	        IF #sUDT_CommonStatus.Manual                                                    // Manual
	        THEN

	            #sUDT_HMIStatus.Status := "DB_HMIStatusConfiguration".Manual;

	        END_IF;

	        IF #sUDT_CommonStatus.ManualRun                                                // Running in manual mode
	        THEN

	            #sUDT_HMIStatus.Status := "DB_HMIStatusConfiguration".ManualRun;

	        END_IF;

	        IF #sUDT_HMIStatus.Specific.DivertsActivationError                             // Divert activation error
	        THEN

	            #sUDT_HMIStatus.Status := "DB_HMIStatusConfiguration".OperationalError;

	        END_IF;

	        IF #sUDT_HMIStatus.Specific.EncoderError                                       // Encoder error
	        THEN

	            #sUDT_HMIStatus.Status := "DB_HMIStatusConfiguration".EncoderError;

	        END_IF;

	        IF #sUDT_HMIStatus.Specific.PEC_EoSJam                                          // IF EOS PEC jam or
	            OR #sUDT_HMIStatus.Specific.PEC_DivertChuteJam                              // Divert chute PEC jam
	            OR #iqUDT_FlowSplitterInterface.InternalErrorPEC                           // Error pec outside of flowsplitter block
	        THEN

	            #sUDT_HMIStatus.Status := "DB_HMIStatusConfiguration".PECJam;

	        END_IF;

	        IF #iqUDT_FlowSplitterInterface.InternalErrorVFD                               // VFD error
	        THEN

	            #sUDT_HMIStatus.Status := "DB_HMIStatusConfiguration".VFDError;

	        END_IF;

	        IF #sUDT_HMIStatus.Specific.Debris                                             // Debris sensor error
	        THEN

	            #sUDT_HMIStatus.Status := "DB_HMIStatusConfiguration".Error;

	        END_IF;

	        IF #sUDT_HMIStatus.Specific.AirPressure                                         // Air pressure error
	        THEN

	            #sUDT_HMIStatus.Status := "DB_HMIStatusConfiguration".Error;

	        END_IF;

	        IF #sUDT_CommonStatus.SafetyStop                                                // Safety stop
	        THEN

	            #sUDT_HMIStatus.Status := "DB_HMIStatusConfiguration".SafetyStop;

	        END_IF;


	        #sUDT_CommonStatusOld := #sUDT_CommonStatus;                                  // Copy status to memory
	        #qUDT_Status := #sUDT_CommonStatus;                                           // Copy status to output

	    END_IF;

	    #qUDT_HMIStatus := #sUDT_HMIStatus;                                           // Copy HMI status to output

	END_REGION

	REGION 11 - Report to control block
	    "FC_EquipmentReport"(iUDT_Status := #sUDT_CommonStatus,                              // Function to manage report between control block and conveyor block
	                         iqUDT_Control := #iqUDT_EquipmentControl);
	END_REGION

	REGION 12 - Internal errors and warnings reset
	    IF #iqUDT_EquipmentControl.Command.Reset
	    THEN
	        #iqUDT_FlowSplitterInterface.InternalErrorPEC := FALSE;
	        #iqUDT_FlowSplitterInterface.InternalWarningTracking := FALSE;
	        #iqUDT_FlowSplitterInterface.InternalErrorTracking := FALSE;
	        #iqUDT_FlowSplitterInterface.InternalWarningVFD := FALSE;
	        #iqUDT_FlowSplitterInterface.InternalErrorVFD := FALSE;
	        #iqUDT_FlowSplitterInterface.ConfigurationError := FALSE;

	    END_IF;
	END_REGION


END_FUNCTION_BLOCK

FUNCTION_BLOCK "FB_G120ForceDormantErrorDetection"
{ S7_Optimized_Access := 'TRUE' }
VERSION : 0.1
// ATTRIBUTES
// AUTO_NUMBER = True
// BLOCK_NUMBER = 212
// END_ATTRIBUTES
   VAR_INPUT
      ix_SystemStopped { ExternalAccessible := 'False'; ExternalVisible := 'False'; ExternalWritable := 'False'} : Bool;   // TRUE = System is stopped
      ix_VFDRunning { ExternalAccessible := 'False'; ExternalVisible := 'False'; ExternalWritable := 'False'} : Bool;   // TRUE = VFD is running
      ix_VFDSTOActive { ExternalAccessible := 'False'; ExternalVisible := 'False'; ExternalWritable := 'False'} : Bool;   // TRUE = STO applied on VFD
      ix_VFDSS1Active { ExternalAccessible := 'False'; ExternalVisible := 'False'; ExternalWritable := 'False'} : Bool;   // TRUE = SS1 applied on VFD
      ix_VFDSLSActive { ExternalAccessible := 'False'; ExternalVisible := 'False'; ExternalWritable := 'False'} : Bool;   // TRUE = SLS applied on VFD
      ix_FDEDMonitoringTimeElaplsed { ExternalAccessible := 'False'; ExternalVisible := 'False'; ExternalWritable := 'False'} : Bool;   // TRUE= Monitoring time in VFD elapsed
   END_VAR

   VAR_IN_OUT
      iqUDT_OuputVFD : "UDT_VfdSiemensPO";
   END_VAR

   VAR
      sx_TestRequired { ExternalAccessible := 'False'; ExternalVisible := 'False'; ExternalWritable := 'False'} : Bool;   // TRUE = Test is required
      sFB_Pulse { ExternalAccessible := 'False'; ExternalVisible := 'False'; ExternalWritable := 'False'; S7_SetPoint := 'False'} : "FB_TimerOnOffDelay";
   END_VAR


BEGIN
	(*
	----------------------------------------------------------------------------------------

	Version history:
	Date        | Version   | Author        | Remark
	----------------------------------------------------------------------------------------
	2020-7-09   | 0.1       | S.Theocharis  | Initial version
	2020-7-14   | 0.2       | Mateusz Piela | Remove timer from the block
	21/02/2023  | 4.0       | F.Baten       | 4.0 Release TIA 17.5
	*)

	REGION Check time

	    //Time to perform test is set to 10 mounth
	    IF #ix_FDEDMonitoringTimeElaplsed
	        AND #ix_SystemStopped
	        AND NOT #ix_VFDRunning
	        AND NOT #ix_VFDSTOActive
	        AND NOT #ix_VFDSS1Active
	        AND NOT #ix_VFDSLSActive
	    THEN
	        #sx_TestRequired := TRUE;
	    END_IF;

	END_REGION

	REGION Trigger Test

	    //create extended pulse for the test signal
	    #sFB_Pulse(iudi_OffDelayTime := 300,
	               ix_SignalToDelay := #sx_TestRequired);

	    //write extended pulse in the test signal
	    #iqUDT_OuputVFD.STW_1.ForceDormantErrorTest := #sFB_Pulse.qx_DelayedSignal;

	    //reset test required trigger and initiate time interval
	    IF #sx_TestRequired
	    THEN
	        #sx_TestRequired := FALSE;
	    END_IF;

	END_REGION
END_FUNCTION_BLOCK

FUNCTION_BLOCK "FB_MCOConveyLinxAixController"
TITLE = FB_VfdConveyLinxAixController
{ S7_Optimized_Access := 'TRUE' }
AUTHOR : Fortna
VERSION : 4.0
//Function to interface with ConveyLinx Aix Controller. On the controller is the possibility to connect two motors with two photoeyes and run the motors independent from each other. Also can each motor output used as a "normal" on/off output
//--V4.0 split the function to accomodate only 1 Motor
   VAR_INPUT
      iUDT_AixConfig { ExternalAccessible := 'False'; ExternalVisible := 'False'; ExternalWritable := 'False'} : "UDT_AixPlcFullControllerConfiguration";   // Configuration structure
      iUDT_AixInputsModule { ExternalAccessible := 'False'; ExternalVisible := 'False'; ExternalWritable := 'False'} : "UDT_AixPlcFullIn";   // ConveyLinxAix inputs structure
      ii_MotorPositionId { ExternalAccessible := 'False'; ExternalVisible := 'False'; ExternalWritable := 'False'} : Int;   // 1 = Master Left, 2 = Master Right, 11 Slave Left, 12 Slave Right
      ii_PositionSetpoint { ExternalAccessible := 'False'; ExternalVisible := 'False'; ExternalWritable := 'False'} : Int;
      ix_24vOk { ExternalAccessible := 'False'; ExternalVisible := 'False'; ExternalWritable := 'False'} : Bool;   // TRUE when 24VDC is healthy
      ix_SimulationModeActive { ExternalAccessible := 'False'; ExternalVisible := 'False'; ExternalWritable := 'False'} : Bool;   // TRUE when Simulation mode active
      ix_StartPositioning { ExternalAccessible := 'False'; ExternalVisible := 'False'; ExternalWritable := 'False'} : Bool;
      ix_ResetPosition { ExternalAccessible := 'False'; ExternalVisible := 'False'; ExternalWritable := 'False'} : Bool;
   END_VAR

   VAR_OUTPUT
      qUDT_HMIStatus { ExternalAccessible := 'False'; ExternalVisible := 'False'; ExternalWritable := 'False'} : "UDT_AixControllerStatus";   // HMI status structure for right motor
      qx_Positioned { ExternalAccessible := 'False'; ExternalVisible := 'False'; ExternalWritable := 'False'} : Bool;
   END_VAR

   VAR_IN_OUT
      iqUDT_AixOutputsModule : "UDT_AixPlcFullOut";   // ConveyLinxAix nr.1 outputs structure
      iqUDT_ConveyorInterface : "UDT_ConveyorInterface";   // Conveyor interface structure Motor
      iqUDT_MCOStatistics : "UDT_VfdStatistics";   // Satistics structure
   END_VAR

   VAR
      sFB_TimerOnOffDelayMCOSpeedFeedbackError { ExternalAccessible := 'False'; ExternalVisible := 'False'; ExternalWritable := 'False'; S7_SetPoint := 'False'} : "FB_TimerOnOffDelay";
      sFB_TimerOnOffDelayCheck24V { ExternalAccessible := 'False'; ExternalVisible := 'False'; ExternalWritable := 'False'; S7_SetPoint := 'False'} : "FB_TimerOnOffDelay";   // MHS "TimerOnOffDelay" - to delay time for MCO 24V contactor
      sFB_TimerOnOffDelayMCO { ExternalAccessible := 'False'; ExternalVisible := 'False'; ExternalWritable := 'False'; S7_SetPoint := 'False'} : "FB_TimerOnOffDelay";
      sFB_TimerOnOffDelayMCOReset { ExternalAccessible := 'False'; ExternalVisible := 'False'; ExternalWritable := 'False'; S7_SetPoint := 'False'} : "FB_TimerOnOffDelay";   // MHS "TimerOnOffDelay" - to extend MCO reset
      sFB_TimerOnOffDelayMCORunningFeedbackError { ExternalAccessible := 'False'; ExternalVisible := 'False'; ExternalWritable := 'False'; S7_SetPoint := 'False'} : "FB_TimerOnOffDelay";
      sFB_TimerOnOffDelayAcceleration { ExternalAccessible := 'False'; ExternalVisible := 'False'; ExternalWritable := 'False'; S7_SetPoint := 'False'} : "FB_TimerOnOffDelay";
      sUDT_HMIStatus { ExternalAccessible := 'False'; ExternalVisible := 'False'; ExternalWritable := 'False'; S7_SetPoint := 'False'} : "UDT_AixControllerStatus";   // Detailed MCO status overview
      sUDT_PNDeviceController { ExternalAccessible := 'False'; ExternalVisible := 'False'; ExternalWritable := 'False'; S7_SetPoint := 'False'} : "UDT_PNDevice";   // PN device info structure, Controller 1
      ss_PNPortsStatusController { ExternalAccessible := 'False'; ExternalVisible := 'False'; ExternalWritable := 'False'} : Array[1..8] of Bool;   // TRUE when specific port has an error, Controller
      sR_TRIG_PNSlaveNotOnline {InstructionName := 'R_TRIG'; LibVersion := '1.0'; ExternalAccessible := 'False'; ExternalVisible := 'False'; ExternalWritable := 'False'; S7_SetPoint := 'False'} : R_TRIG;   // Rising edge for trigger Profinet slave not online statistics
      sR_TRIG_PNSlaveError {InstructionName := 'R_TRIG'; LibVersion := '1.0'; ExternalAccessible := 'False'; ExternalVisible := 'False'; ExternalWritable := 'False'; S7_SetPoint := 'False'} : R_TRIG;   // Rising edge for trigger Profinet slave error statistics
      sR_TRIG_MCOInternalError {InstructionName := 'R_TRIG'; LibVersion := '1.0'; ExternalAccessible := 'False'; ExternalVisible := 'False'; ExternalWritable := 'False'; S7_SetPoint := 'False'} : R_TRIG;   // Rising edge for trigger Internal MCO Error statistics
      sR_TRIG_Running {InstructionName := 'R_TRIG'; LibVersion := '1.0'; ExternalAccessible := 'False'; ExternalVisible := 'False'; ExternalWritable := 'False'; S7_SetPoint := 'False'} : R_TRIG;   // Rising edge for trigger running motor
      sR_TRIG_CommunicationErrorMCO {InstructionName := 'R_TRIG'; LibVersion := '1.0'; ExternalAccessible := 'False'; ExternalVisible := 'False'; ExternalWritable := 'False'; S7_SetPoint := 'False'} : R_TRIG;   // Rising edge for trigger communication error
      sR_TRIG_ResetPosition {InstructionName := 'R_TRIG'; LibVersion := '1.0'; ExternalAccessible := 'False'; ExternalVisible := 'False'; ExternalWritable := 'False'; S7_SetPoint := 'False'} : R_TRIG;   // Rising edge reset position
      sF_TRIG_RunFwd {InstructionName := 'F_TRIG'; LibVersion := '1.0'; ExternalAccessible := 'False'; ExternalVisible := 'False'; ExternalWritable := 'False'; S7_SetPoint := 'False'} : F_TRIG;   // Falling edge for run forward signal
      sF_TRIG_RunRvs {InstructionName := 'F_TRIG'; LibVersion := '1.0'; ExternalAccessible := 'False'; ExternalVisible := 'False'; ExternalWritable := 'False'; S7_SetPoint := 'False'} : F_TRIG;   // Falling edge for run reverse signal
      sr_ActualSpeedSetpoint { ExternalAccessible := 'False'; ExternalVisible := 'False'; ExternalWritable := 'False'} : Real;   // Actual speed setpoint motor
      si_ActualSpeed { ExternalAccessible := 'False'; ExternalVisible := 'False'; ExternalWritable := 'False'} : Int;   // Actual speed motor
      si_MotorAcceleration { ExternalAccessible := 'False'; ExternalVisible := 'False'; ExternalWritable := 'False'} : Int;   // Left motor acceleration
      si_MotorDeceleration { ExternalAccessible := 'False'; ExternalVisible := 'False'; ExternalWritable := 'False'} : Int;   // Motor deceleration
      si_LeftMotorPosition { ExternalAccessible := 'False'; ExternalVisible := 'False'; ExternalWritable := 'False'} : Int;   // Left motor actual position
      si_LastLeftMotorPosition { ExternalAccessible := 'False'; ExternalVisible := 'False'; ExternalWritable := 'False'} : Int;   // Left motor last cycle position
      si_RightMotorPosition { ExternalAccessible := 'False'; ExternalVisible := 'False'; ExternalWritable := 'False'} : Int;   // Right motor actual position
      si_LastRightMotorPosition { ExternalAccessible := 'False'; ExternalVisible := 'False'; ExternalWritable := 'False'} : Int;   // Right motor last cycle position
      sx_GeneralStatisticsReset { ExternalAccessible := 'False'; ExternalVisible := 'False'; ExternalWritable := 'False'} : Bool;   // Reset from or right conveyor
      sx_HardwareOK { ExternalAccessible := 'False'; ExternalVisible := 'False'; ExternalWritable := 'False'} : Bool;   // Hardware is ok
      sx_ConfigurationError { ExternalAccessible := 'False'; ExternalVisible := 'False'; ExternalWritable := 'False'} : Bool;   // Commissioning: configuration error
      sx_PNDeviceHealthyControler { ExternalAccessible := 'False'; ExternalVisible := 'False'; ExternalWritable := 'False'} : Bool;   // Profinet device is online and error free, Controller 1
      sx_AixAvailableControler { ExternalAccessible := 'False'; ExternalVisible := 'False'; ExternalWritable := 'False'} : Bool;   // Hardware of MCO is ok and no communication error with movikit, Controller 1
      sx_24vOk { ExternalAccessible := 'False'; ExternalVisible := 'False'; ExternalWritable := 'False'} : Bool;   // 24VDC is healthy
      sx_ErrorActive { ExternalAccessible := 'False'; ExternalVisible := 'False'; ExternalWritable := 'False'} : Bool;   // Block has an error
      sx_EnableOperation { ExternalAccessible := 'False'; ExternalVisible := 'False'; ExternalWritable := 'False'} : Bool;   // Enable operation signal
      sx_RunForward { ExternalAccessible := 'False'; ExternalVisible := 'False'; ExternalWritable := 'False'} : Bool;   // Start MCO forward
      sx_RunReverse { ExternalAccessible := 'False'; ExternalVisible := 'False'; ExternalWritable := 'False'} : Bool;   // Start MCO backward
      sx_SpeedSetpointReached { ExternalAccessible := 'False'; ExternalVisible := 'False'; ExternalWritable := 'False'} : Bool;   // Speed setpoint reached motor
      sx_SpeedFeedbackError { ExternalAccessible := 'False'; ExternalVisible := 'False'; ExternalWritable := 'False'} : Bool;   // motor speed feedback error
      sx_ErrorController { ExternalAccessible := 'False'; ExternalVisible := 'False'; ExternalWritable := 'False'} : Bool;   // Active if any erorr from controller 1 is active
      sx_ErrorCMotor { ExternalAccessible := 'False'; ExternalVisible := 'False'; ExternalWritable := 'False'} : Bool;   // TRUE if error from controler motor is active
      sx_Accelerating { ExternalAccessible := 'False'; ExternalVisible := 'False'; ExternalWritable := 'False'} : Bool;   // Motor acceleration
      sx_HardwareOk_Motor { ExternalAccessible := 'False'; ExternalVisible := 'False'; ExternalWritable := 'False'} : Bool;   // Motor hardware ok
      sx_LeftServoHomeHasBeenSet { ExternalAccessible := 'False'; ExternalVisible := 'False'; ExternalWritable := 'False'} : Bool;   // Servo position has beeen reset to 0
      sx_RightServoHomeHasBeenSet { ExternalAccessible := 'False'; ExternalVisible := 'False'; ExternalWritable := 'False'} : Bool;   // Servo position has beeen reset to 0
      sb_MotorRotationStatus { ExternalAccessible := 'False'; ExternalVisible := 'False'; ExternalWritable := 'False'} : Byte;   // 0 Motor not running, Normal or Servo Braking Mode applied; 1 Motor running in CCW Direction; 2 Motor running in CW Direction; 3 Motor not running and Free Braking Mode applied
   END_VAR

   VAR CONSTANT
      ci_MCOArea : UInt := 1;   // Area ID of IO Profinet devices
      ci_SubmoduleHWType : UInt := 5;   // Submodule HW_type number
      ci_TelegramSlot : UInt := 1;   // Free Siemens telegram slot
      ci_TelegramSubslot : UInt := 3;   // Free Siemens telegram subslot
      ci_NumberOfProfinetPorts : Int := 2;   // Number of Profinet ports in device
      cr_MaximumOutput : Real := 16384.0;   // PLC maximum output value
      cw_ActualSpeedMask : Word := 2#0011_1111_1111_1111;   // Mask to get the speed from the profinet MotorActualSpeed Word
      cudi_ExtendedResetTime : UDInt := 500;   // Extending the reset puls
      cudi_HardwareCheckDelay : UDInt := 2000;   // Delay to enable hardware to start up, checking will start after this time
      cudi_FeedbackErrorDelay : UDInt := 10000;   // Maximum delaytime deviation from setpoint is allowed
      cudi_TimeOffsetSpeedmonitoring : UDInt := 2000;   // Additional time
      cudi_HeartbeatDelay : UDInt := 5000;   // Maximum dely between heartbeat
      ci_Master_Left : Int := 1;
      ci_Master_Right : Int := 2;
      ci_Slave_Left : Int := 11;
      ci_Slave_Right : Int := 12;
   END_VAR


BEGIN
	(*
	----------------------------------------------------------------------------------------

	Version history:
	Date        | Version   | Author        | Remark
	----------------------------------------------------------------------------------------
	03/01/2022  | 1.0       | N.Kadam       | First release MHSE TIA 16.0
	24/03/2022  | 1.1       | M.Piela       | Bug fix, adding running feedback error
	05/05/2022  | 1.2       | M.Piela       | Status update
	31/05/2022  | 1.3       | M.Piela       | Ramp up/down calculation fix
	21/07/2022  | 1.4       | M.Piela       | Prevent motor to go below the minimum speed
	29/07/2022  | 1.5       | M.Piela       | Status update, add hardware ok to the profinet checking
	01/08/2022  | 1.6       | M.Piela       | Add Hardware ok to reset internal error
	01/08/2022  | 1.7       | G.Vlooswijk   | Fix to make it possible to run 1 of the 2 motors
	                                        | Check setpoint instead of sx_EnableOperation for Feedback Error check
	                                        | Removed if statement i_UDT_Ai2Config.DirectionReversal, speed from controller always positive
	06/08/2022  | 1.8       | G.Vlooswijk   | Removed minimal speedsetpoint
	05/07/2023  | 1.9       | F.Baten       | Complete separation of 2 motors
	13/09/2023  | 4.0       | F.Baten       | Reorganised structure and took out unused symbolics
	                                        | Status as 1 controller with 2 seperate controlled motors
	02/05/2024  | 5.0       | I.Ajram       | Split the function to accomodate only 1 Motor, added an input to indicate which motor to control
	08/05/2024  | 5.1       | S.Nieswiec    | qUDT_AixOutputsModule move to in/out variables, name changed to iqUDT_AixOutputsModule
	08/05/2024  | 5.2       | K. Pokorski   | Add displacement calculation
	13/05/2024  | 5.3       | K. Pokorski   | Add roller ratio
	08/06/2024  | 5.4       | S.Nieswiec    | Fixed servo delta calculation (went back to previous functioning version), adjusted region numbering
	                                        | displacement was negative on some conveyors while positive on others
	21/06/2024  | 5.5       | I.Ajram       | Added Master / Slave Mod, Slave is used when one conveyor is controlling more than 1 MCO, the rest will act/ be configured as slaves
	*)

	REGION 1 - Get Device Profinet information

	    //Get Device Profinet name, Controller
	    "FC_GetDevicePN"(is_PNDeviceName := #iUDT_AixConfig.AixContrlPNDeviceName,
	                     ix_SimulationModeActive := #ix_SimulationModeActive,
	                     iqUDT_PND := #sUDT_PNDeviceController);

	    //Get number of ports, Controller
	    "FC_GetPNPortStatus"(ii_NumberOfPorts := #ci_NumberOfProfinetPorts,
	                         iUDT_DevicePNInfo := #sUDT_PNDeviceController,
	                         qa_PortFault => #ss_PNPortsStatusController);

	END_REGION

	REGION 2 - Reset errors


	    REGION 2.1 - Motor

	        // Reset errors when InternalErrorReset is given
	        IF #iqUDT_ConveyorInterface.InternalErrorReset OR (NOT #iqUDT_ConveyorInterface.HardwareOk AND #sUDT_HMIStatus.PNSlaveNotOnline)
	        THEN
	            #sUDT_HMIStatus.PNSlaveNotOnline := FALSE;
	            #sUDT_HMIStatus.PNSlaveError := FALSE;
	            #sUDT_HMIStatus.InternalError := FALSE;
	            #sUDT_HMIStatus.PNSlaveWarning := FALSE;
	            #sUDT_HMIStatus.SpeedFeedbackError := FALSE;
	            #sx_SpeedFeedbackError := FALSE;
	            #sx_ErrorCMotor := FALSE;
	            #sUDT_HMIStatus.MotorStatus.Overheat := FALSE;
	            #sUDT_HMIStatus.MotorStatus.MaxTorque := FALSE;
	            #sUDT_HMIStatus.MotorStatus.ShortCircuit := FALSE;
	            #sUDT_HMIStatus.MotorStatus.MotorNotConnected := FALSE;
	            #sUDT_HMIStatus.MotorStatus.Overload := FALSE;
	            #sUDT_HMIStatus.MotorStatus.Stalled := FALSE;
	            #sUDT_HMIStatus.MotorStatus.BadHall := FALSE;
	            #sUDT_HMIStatus.MotorStatus.BoardOverheat := FALSE;
	            #sUDT_HMIStatus.MotorStatus.OverVoltage := FALSE;
	            #sUDT_HMIStatus.MotorStatus.LowVoltage := FALSE;
	            #iqUDT_ConveyorInterface.InternalErrorVFD := FALSE;

	        END_IF;

	    END_REGION

	    REGION 2.2 - Reset pulse
	        // Create extended pulse for MCO Reset
	        #sFB_TimerOnOffDelayMCOReset(iudi_OnDelayTime := #cudi_ExtendedResetTime,
	                                     iudi_OffDelayTime := 0,
	                                     ix_SignalToDelay := #iqUDT_AixOutputsModule.ClearMotorError = 1,
	                                     ix_Enable := TRUE);
	        // set the reset signal directly when reset is active
	        IF #iqUDT_ConveyorInterface.InternalErrorReset THEN
	            #iqUDT_AixOutputsModule.ClearMotorError := 1;
	        END_IF;

	        // Reset the ClearMotorError after 500[ms] pulse
	        IF #sFB_TimerOnOffDelayMCOReset.qx_DelayedSignal
	        THEN
	            #iqUDT_AixOutputsModule.ClearMotorError := 0;
	        END_IF;

	    END_REGION

	END_REGION

	REGION 3 - Hardware checks

	    // Hardware will only be available after the delay, so the device has time for the initialisation
	    #sFB_TimerOnOffDelayCheck24V(iudi_OnDelayTime := #cudi_HardwareCheckDelay,
	                                 ix_SignalToDelay := #ix_24vOk);

	    #sx_24vOk := #sFB_TimerOnOffDelayCheck24V.qx_DelayedSignal;

	    #sx_HardwareOk_Motor := #iqUDT_ConveyorInterface.HardwareOk AND #iUDT_AixConfig.Motor.MotorExist;

	    #sx_HardwareOK := NOT #ix_SimulationModeActive
	    AND #sx_24vOk
	    AND (#sx_HardwareOk_Motor OR NOT #iUDT_AixConfig.Motor.MotorExist)
	    AND (#ss_PNPortsStatusController[1] OR #ss_PNPortsStatusController[2])
	    AND #iqUDT_ConveyorInterface.HardwareOk;


	    // Check if PN device is online
	    IF NOT "DB_ProfinetDiagnostic".ProfinetNetworks[#sUDT_PNDeviceController.PNNetworknumber].DeviceStatus[#sUDT_PNDeviceController.PNDeviceNumber].DeviceState.Exist
	        AND #sx_HardwareOK
	    THEN
	        #sUDT_HMIStatus.PNSlaveNotOnline := TRUE;
	    END_IF;

	    // Check IF PN ports are healthy
	    IF #ss_PNPortsStatusController[1] XOR #ss_PNPortsStatusController[2]

	    THEN
	        #sUDT_HMIStatus.PNSlaveWarning := TRUE;
	    END_IF;

	    // Check if PN device has an error
	    IF "DB_ProfinetDiagnostic".ProfinetNetworks[#sUDT_PNDeviceController.PNNetworknumber].DeviceStatus[#sUDT_PNDeviceController.PNDeviceNumber].DeviceState.Error
	        AND #sx_HardwareOK
	        AND NOT #sUDT_HMIStatus.PNSlaveWarning
	    THEN
	        #sUDT_HMIStatus.PNSlaveError := TRUE;
	    END_IF;

	    // Set bit when PN device is healthy (online and no error)
	    #sx_PNDeviceHealthyControler := NOT #sUDT_HMIStatus.PNSlaveNotOnline
	    AND NOT #sUDT_HMIStatus.PNSlaveError
	    AND #sUDT_PNDeviceController.PNDeviceFound
	    AND #sx_24vOk;

	    // Set hardware available bit when all conditions are met
	    #sx_AixAvailableControler := (#sx_24vOk
	    AND #sx_PNDeviceHealthyControler
	    AND (#sx_HardwareOk_Motor OR NOT #iUDT_AixConfig.Motor.MotorExist))
	    OR #ix_SimulationModeActive;

	    // Check communication (heartbeat)
	    #sFB_TimerOnOffDelayMCO(iudi_OnDelayTime := #cudi_HeartbeatDelay,
	                            ix_SignalToDelay := NOT #iUDT_AixInputsModule.AllSensorPortInputs.Heartbeat);

	    // Set error when MoviKit communication is not available
	    IF #sFB_TimerOnOffDelayMCO.qx_DelayedSignal AND #sx_HardwareOK
	    THEN

	        #sUDT_HMIStatus.CommunicationErrorVFD := TRUE;

	    END_IF;
	END_REGION

	REGION 4 - Check errors and warnings
	    REGION 4.1 - Error from controller for right motor
	        IF #ii_MotorPositionId = #ci_Master_Right OR #ii_MotorPositionId = #ci_Slave_Right THEN
	            //Write errors to UDT_Status
	            IF #iUDT_AixInputsModule.RightMotorDiagnostic.Overheat
	            THEN
	                #sUDT_HMIStatus.MotorStatus.Overheat := TRUE;
	            END_IF;

	            #sUDT_HMIStatus.MotorStatus.MaxTorque := #iUDT_AixInputsModule.RightMotorDiagnostic.MaxTorque;

	            IF #iUDT_AixInputsModule.RightMotorDiagnostic.ShortCircuit
	            THEN
	                #sUDT_HMIStatus.MotorStatus.ShortCircuit := TRUE;
	            END_IF;

	            IF #iUDT_AixInputsModule.RightMotorDiagnostic.MotorNotConnected
	            THEN
	                #sUDT_HMIStatus.MotorStatus.MotorNotConnected := TRUE;
	            END_IF;

	            IF #iUDT_AixInputsModule.RightMotorDiagnostic.Overload
	            THEN
	                #sUDT_HMIStatus.MotorStatus.Overload := TRUE;
	            END_IF;

	            IF #iUDT_AixInputsModule.RightMotorDiagnostic.Stalled
	            THEN
	                #sUDT_HMIStatus.MotorStatus.Stalled := TRUE;
	            END_IF;

	            IF #iUDT_AixInputsModule.RightMotorDiagnostic.BadHall
	            THEN
	                #sUDT_HMIStatus.MotorStatus.BadHall := TRUE;
	            END_IF;

	            IF #iUDT_AixInputsModule.RightMotorDiagnostic.BoardOverheat
	            THEN
	                #sUDT_HMIStatus.MotorStatus.BoardOverheat := TRUE;
	            END_IF;

	            IF #iUDT_AixInputsModule.RightMotorDiagnostic.OverVoltage
	            THEN
	                #sUDT_HMIStatus.MotorStatus.OverVoltage := TRUE;
	            END_IF;

	            IF #iUDT_AixInputsModule.RightMotorDiagnostic.LowVoltage
	            THEN
	                #sUDT_HMIStatus.MotorStatus.LowVoltage := TRUE;
	            END_IF;

	        END_IF;
	    END_REGION

	    REGION 4.2 - Error from controller for left motor
	        IF #ii_MotorPositionId = #ci_Master_Left OR #ii_MotorPositionId = #ci_Slave_Left THEN
	            //Write errors to UDT_Status
	            IF #iUDT_AixInputsModule.LeftMotorDiagnostic.Overheat
	            THEN
	                #sUDT_HMIStatus.MotorStatus.Overheat := TRUE;
	            END_IF;

	            #sUDT_HMIStatus.MotorStatus.MaxTorque := #iUDT_AixInputsModule.LeftMotorDiagnostic.MaxTorque;

	            IF #iUDT_AixInputsModule.LeftMotorDiagnostic.ShortCircuit
	            THEN
	                #sUDT_HMIStatus.MotorStatus.ShortCircuit := TRUE;
	            END_IF;

	            IF #iUDT_AixInputsModule.LeftMotorDiagnostic.MotorNotConnected
	            THEN
	                #sUDT_HMIStatus.MotorStatus.MotorNotConnected := TRUE;
	            END_IF;

	            IF #iUDT_AixInputsModule.LeftMotorDiagnostic.Overload
	            THEN
	                #sUDT_HMIStatus.MotorStatus.Overload := TRUE;
	            END_IF;

	            IF #iUDT_AixInputsModule.LeftMotorDiagnostic.Stalled
	            THEN
	                #sUDT_HMIStatus.MotorStatus.Stalled := TRUE;
	            END_IF;

	            IF #iUDT_AixInputsModule.LeftMotorDiagnostic.BadHall
	            THEN
	                #sUDT_HMIStatus.MotorStatus.BadHall := TRUE;
	            END_IF;

	            IF #iUDT_AixInputsModule.LeftMotorDiagnostic.BoardOverheat
	            THEN
	                #sUDT_HMIStatus.MotorStatus.BoardOverheat := TRUE;
	            END_IF;

	            IF #iUDT_AixInputsModule.LeftMotorDiagnostic.OverVoltage
	            THEN
	                #sUDT_HMIStatus.MotorStatus.OverVoltage := TRUE;
	            END_IF;

	            IF #iUDT_AixInputsModule.LeftMotorDiagnostic.LowVoltage
	            THEN
	                #sUDT_HMIStatus.MotorStatus.LowVoltage := TRUE;
	            END_IF;
	        END_IF;
	    END_REGION

	    REGION 4.3 - Collective Error
	        //If any error from controller motor ocursed then set error to TRUE
	        IF #iUDT_AixConfig.Motor.MotorExist
	        THEN
	            #sx_ErrorCMotor := #sUDT_HMIStatus.MotorStatus.Overheat OR
	            // #sUDT_HMIStatus.MotorError.MaxTorque OR
	            #sUDT_HMIStatus.MotorStatus.ShortCircuit OR
	            #sUDT_HMIStatus.MotorStatus.MotorNotConnected OR
	            #sUDT_HMIStatus.MotorStatus.Overload OR
	            #sUDT_HMIStatus.MotorStatus.Stalled OR
	            #sUDT_HMIStatus.MotorStatus.BadHall OR
	            #sUDT_HMIStatus.MotorStatus.BoardOverheat OR
	            #sUDT_HMIStatus.MotorStatus.OverVoltage OR
	            #sUDT_HMIStatus.MotorStatus.LowVoltage OR
	            #sUDT_HMIStatus.SpeedFeedbackError OR
	            #sUDT_HMIStatus.PNSlaveNotOnline OR
	            #sUDT_HMIStatus.PNSlaveError;
	        END_IF;
	    END_REGION

	    REGION 4.4 - Controller general

	        // Error Controller is two drives combined
	        #sx_ErrorController :=
	        #iUDT_AixInputsModule.ConveyStopStatus.StopActiveLostConn OR
	        #iUDT_AixInputsModule.ConveyStopStatus.StopActiveLostPLC OR
	        #sx_ErrorCMotor OR
	        FALSE;

	        // Check if a Controller has an error
	        #sx_ErrorActive := (#sx_ErrorController AND #iUDT_AixConfig.Motor.MotorExist)
	        OR #sFB_TimerOnOffDelayMCORunningFeedbackError.qx_DelayedSignal
	        OR #sFB_TimerOnOffDelayMCOSpeedFeedbackError.qx_DelayedSignal;

	        // Internal error
	        #sUDT_HMIStatus.InternalError := #sx_AixAvailableControler AND #sx_ErrorController;

	    END_REGION

	END_REGION

	REGION 5 - Check if configuration is ok for commissioning purposes

	    IF (
	        #iUDT_AixConfig.Motor.MotorExist                            // Check only if motor exists
	        AND (#iUDT_AixConfig.Motor.RampUpTime > 0)                  // If ramp up time is greater than 0
	        AND (#iUDT_AixConfig.Motor.RampDownTime > 0)                // and ramp down time is greater than 0
	        )
	        AND
	        (
	        #sUDT_PNDeviceController.PNDeviceFound
	        OR NOT #iUDT_AixConfig.Motor.MotorExist                       // and device found in PN structure
	        OR #ix_SimulationModeActive                                 // or simulation mode is active
	        )
	    THEN
	        #sx_ConfigurationError := FALSE;                                // Reset configuration error
	    ELSE
	        #sx_ConfigurationError := TRUE;                                 // Set configuration error
	    END_IF;

	END_REGION

	REGION 6 - Prepare output data for Controller

	    REGION 6.1 - Set direction for motor

	        // If Run forward is requested, set direction to forward
	        IF #iqUDT_ConveyorInterface.RunFwd
	            AND #iUDT_AixConfig.Motor.InterlockFwd
	        THEN
	            #sx_RunForward := TRUE;
	            #sx_RunReverse := FALSE;
	        END_IF;

	        // If Run reverse is requested, set direction into reverse
	        IF #iqUDT_ConveyorInterface.RunRvs
	            AND #iUDT_AixConfig.Motor.InterlockRvs
	        THEN
	            #sx_RunReverse := TRUE;
	            #sx_RunForward := FALSE;
	        END_IF;

	    END_REGION


	    REGION 6.3 - Stopping motor

	        // Create trigger when direction signal falling
	        #sF_TRIG_RunFwd(CLK := #iqUDT_ConveyorInterface.RunFwd);
	        #sF_TRIG_RunRvs(CLK := #iqUDT_ConveyorInterface.RunRvs);

	        // When no run signal is given the controllers should stop
	        IF (NOT #iqUDT_ConveyorInterface.RunRvs AND NOT #iqUDT_ConveyorInterface.RunFwd)
	            OR (#iqUDT_ConveyorInterface.RunRvs AND #iqUDT_ConveyorInterface.RunFwd)
	            OR (#sF_TRIG_RunRvs.Q)
	            OR (#sF_TRIG_RunFwd.Q)
	            OR #sx_ErrorActive
	        THEN
	            #sx_RunReverse := FALSE;
	            #sx_RunForward := FALSE;
	        END_IF;

	    END_REGION

	    REGION 6.5 - Check for enable operation signal

	        //Enable operation if there is no error active and there is an given direction
	        #sx_EnableOperation := NOT #sx_ErrorActive
	        AND NOT #sx_ConfigurationError
	        AND (#sx_RunForward OR #sx_RunReverse);
	    END_REGION

	    REGION 6.6 - Calculate acceleration and deceleration values

	        //Motor
	        //Recalculating Acceleration (from ms to mm)
	        #si_MotorAcceleration := REAL_TO_INT((INT_TO_REAL(#iqUDT_ConveyorInterface.SpeedSetpoint) * #iUDT_AixConfig.Motor.Ratio / 2) * (UDINT_TO_REAL(#iUDT_AixConfig.Motor.RampUpTime) / 1000));

	        //Recalculating Deceleration (from ms to mm)
	        #si_MotorDeceleration := REAL_TO_INT((INT_TO_REAL(#iqUDT_ConveyorInterface.SpeedSetpoint) * #iUDT_AixConfig.Motor.Ratio / 2) * (UDINT_TO_REAL(#iUDT_AixConfig.Motor.RampDownTime) / 1000));

	    END_REGION

	END_REGION

	REGION 7 - Write outputs to controller
	    // Clear speed setpoint when no run request or above direction request or is configuration error
	    IF #sx_EnableOperation
	    THEN
	        #sr_ActualSpeedSetpoint := INT_TO_REAL(#iqUDT_ConveyorInterface.SpeedSetpoint) / #iUDT_AixConfig.Motor.Ratio;
	    ELSE
	        #sr_ActualSpeedSetpoint := 0;
	    END_IF;

	    REGION 7.1 - Controller Left motor

	        IF #ii_MotorPositionId = #ci_Master_Left OR #ii_MotorPositionId = #ci_Slave_Left THEN
	            //Seting up speed for Left motor
	            #iqUDT_AixOutputsModule.LeftSetMotorSpeed := REAL_TO_INT(#sr_ActualSpeedSetpoint);
	            IF #iqUDT_AixOutputsModule.LeftSetMotorSpeed > #cr_MaximumOutput
	            THEN
	                // if actual value is greater than maximmu output value then write maximmu output value
	                #iqUDT_AixOutputsModule.LeftSetMotorSpeed := REAL_TO_INT(#cr_MaximumOutput);
	            END_IF;

	            //Check if motor is in use, if yes set parameters from conveyor to the controller and motor
	            IF #iUDT_AixConfig.Motor.MotorExist
	            THEN
	                //Setting up run bit, acceleration, deceleration
	                #iqUDT_AixOutputsModule.LeftMotorControl.Run := #sx_EnableOperation
	                AND (#iqUDT_ConveyorInterface.RunFwd OR #iqUDT_ConveyorInterface.RunRvs);

	                // Position setpoint
	                #iqUDT_AixOutputsModule.ServoControlDistanceLeft := #ii_PositionSetpoint;

	                //Start positioning
	                #iqUDT_AixOutputsModule.ServoControlCommandLeft.%X1 := #ix_StartPositioning
	                AND #sx_EnableOperation
	                AND (#iqUDT_ConveyorInterface.RunFwd OR #iqUDT_ConveyorInterface.RunRvs);

	                // Reset position
	                #sR_TRIG_ResetPosition(CLK := #ix_ResetPosition);

	                // Reset position after every operation
	                IF #sR_TRIG_ResetPosition.Q THEN

	                    #iqUDT_AixOutputsModule.ServoControlCommandLeft.%X0 := TRUE;

	                END_IF;

	                // End homing procedure when motor is reset
	                IF #iUDT_AixInputsModule.ServoStatusLeft.%X1 THEN

	                    #iqUDT_AixOutputsModule.ServoControlCommandLeft.%X0 := FALSE;

	                END_IF;


	                #iqUDT_AixOutputsModule.LeftSetMotorAccel := #si_MotorAcceleration;
	                #iqUDT_AixOutputsModule.LeftSetMotorDeccel := #si_MotorDeceleration;

	                //Setting direction
	                IF (#sx_RunReverse AND NOT #iUDT_AixConfig.Motor.DirectionReversal)
	                    OR (#sx_RunForward AND #iUDT_AixConfig.Motor.DirectionReversal)
	                THEN
	                    #iqUDT_AixOutputsModule.LeftMotorControl.MotorDirection := 1;
	                ELSE
	                    #iqUDT_AixOutputsModule.LeftMotorControl.MotorDirection := 0;
	                END_IF;
	            ELSE
	                #iqUDT_AixOutputsModule.LeftMotorControl.Run := FALSE;
	            END_IF;
	        END_IF;
	    END_REGION

	    REGION 7.2 - Controller right motor
	        IF #ii_MotorPositionId = #ci_Master_Right OR #ii_MotorPositionId = #ci_Slave_Right THEN
	            //Seting up speed for Right motor
	            #iqUDT_AixOutputsModule.RightSetMotorSpeed := REAL_TO_INT(#sr_ActualSpeedSetpoint);
	            IF #iqUDT_AixOutputsModule.RightSetMotorSpeed > #cr_MaximumOutput
	            THEN
	                // if actual value is greater than maximmu output value then write maximmu output value
	                #iqUDT_AixOutputsModule.RightSetMotorSpeed := REAL_TO_INT(#cr_MaximumOutput);
	            END_IF;

	            //Check if motor is in use, if yes set parameters from conveyor to the controller and motor
	            IF #iUDT_AixConfig.Motor.MotorExist
	            THEN
	                //Setting up run bit, acceleration, deceleration
	                #iqUDT_AixOutputsModule.RightMotorControl.Run := #sx_EnableOperation
	                AND (#iqUDT_ConveyorInterface.RunFwd OR #iqUDT_ConveyorInterface.RunRvs);

	                // Position setpoint
	                #iqUDT_AixOutputsModule.ServoControlDistanceRight := #ii_PositionSetpoint;

	                //Start positioning
	                #iqUDT_AixOutputsModule.ServoControlCommandRight.%X1 := #ix_StartPositioning
	                AND #sx_EnableOperation
	                AND (#iqUDT_ConveyorInterface.RunFwd OR #iqUDT_ConveyorInterface.RunRvs);

	                // Reset position
	                #sR_TRIG_ResetPosition(CLK := #ix_ResetPosition);

	                // Reset position after every operation
	                IF #sR_TRIG_ResetPosition.Q THEN

	                    #iqUDT_AixOutputsModule.ServoControlCommandRight.%X0 := TRUE;

	                END_IF;

	                // End homing procedure when motor is reset
	                IF #iUDT_AixInputsModule.ServoStatusRight.%X1 THEN

	                    #iqUDT_AixOutputsModule.ServoControlCommandRight.%X0 := FALSE;

	                END_IF;


	                #iqUDT_AixOutputsModule.RightSetMotorAccel := #si_MotorAcceleration;
	                #iqUDT_AixOutputsModule.RightSetMotorDeccel := #si_MotorDeceleration;

	                //Setting direction
	                IF (#sx_RunReverse AND NOT #iUDT_AixConfig.Motor.DirectionReversal)
	                    OR (#sx_RunForward AND #iUDT_AixConfig.Motor.DirectionReversal)
	                THEN
	                    #iqUDT_AixOutputsModule.RightMotorControl.MotorDirection := 1;
	                ELSE
	                    #iqUDT_AixOutputsModule.RightMotorControl.MotorDirection := 0;
	                END_IF;
	            ELSE
	                #iqUDT_AixOutputsModule.RightMotorControl.Run := FALSE;
	            END_IF;
	        END_IF;
	    END_REGION

	END_REGION

	REGION 8 - Reading actual speed

	    REGION 8.1 - Left Motor
	        IF #ii_MotorPositionId = #ci_Master_Left OR #ii_MotorPositionId = #ci_Slave_Left THEN
	            //When motors are in constant speed use motor actual speed
	            IF #iUDT_AixConfig.Motor.MotorExist
	            THEN
	                #si_ActualSpeed := REAL_TO_INT(INT_TO_REAL(WORD_TO_INT(#iUDT_AixInputsModule.LeftMotorActualSpeed & #cw_ActualSpeedMask)) * #iUDT_AixConfig.Motor.Ratio);
	            ELSE
	                #si_ActualSpeed := 0;
	            END_IF;
	        END_IF;
	    END_REGION

	    REGION 8.2 - Right Motor
	        IF #ii_MotorPositionId = #ci_Master_Right OR #ii_MotorPositionId = #ci_Slave_Right THEN
	            //When motors are in constant speed use motor actual speed
	            IF #iUDT_AixConfig.Motor.MotorExist
	            THEN
	                #si_ActualSpeed := REAL_TO_INT(INT_TO_REAL(WORD_TO_INT(#iUDT_AixInputsModule.RightMotorActualSpeed & #cw_ActualSpeedMask)) * #iUDT_AixConfig.Motor.Ratio);
	            ELSE
	                #si_ActualSpeed := 0;
	            END_IF;
	        END_IF;
	    END_REGION

	    REGION 8.3 - Calculation
	        //Actual speed is in mm/s
	        //Sets error signal if an motor is running for a longer time with a diferent speed than speed setpoint but after a certain time
	        #sFB_TimerOnOffDelayMCORunningFeedbackError(iudi_OnDelayTime := #cudi_FeedbackErrorDelay,
	                                                    ix_SignalToDelay := #sr_ActualSpeedSetpoint <> 0.0 AND NOT (#si_ActualSpeed <> 0));

	        //The motor should start running after specific time. If not the MCORunningFeedback error occured
	        #sFB_TimerOnOffDelayMCOSpeedFeedbackError(iudi_OnDelayTime := #cudi_FeedbackErrorDelay,
	                                                  ix_SignalToDelay := #sx_SpeedFeedbackError);

	        IF #sFB_TimerOnOffDelayMCORunningFeedbackError.qx_DelayedSignal OR #sFB_TimerOnOffDelayMCOSpeedFeedbackError.qx_DelayedSignal
	        THEN
	            #sUDT_HMIStatus.SpeedFeedbackError := TRUE;
	        END_IF;

	        //Sets signal for the time in which the motors are accelerating
	        #sFB_TimerOnOffDelayAcceleration(iudi_OnDelayTime := 0,
	                                         iudi_OffDelayTime := #iUDT_AixConfig.Motor.RampUpTime + #cudi_TimeOffsetSpeedmonitoring,
	                                         ix_SignalToDelay := #sR_TRIG_Running.Q,
	                                         ix_Enable := TRUE,
	                                         qx_DelayedSignal => #sx_Accelerating);


	        //If conveyor is running and runs forwad or backwards and is not accelerating, when any motor is running at a lower/greater speed than set speed then set an error
	        IF #iqUDT_ConveyorInterface.VFDRunning AND (#iqUDT_ConveyorInterface.RunFwd OR #iqUDT_ConveyorInterface.RunRvs) AND NOT #sx_Accelerating
	        THEN
	            //Check if the difference betwen acctual speed and set speed is bigger than deviation then set error
	            #sx_SpeedFeedbackError := #iUDT_AixConfig.Motor.SpeedSetpointWindow < (ABS(#si_ActualSpeed) - (#iqUDT_ConveyorInterface.SpeedSetpoint));
	        END_IF;


	        // Check IF speed setpoint is reached FOR motor
	        #sx_SpeedSetpointReached := (ABS(#si_ActualSpeed) >= ((#iqUDT_ConveyorInterface.SpeedSetpoint) - #iUDT_AixConfig.Motor.SpeedSetpointWindow))
	        AND (ABS(#si_ActualSpeed) <= ((#iqUDT_ConveyorInterface.SpeedSetpoint) + #iUDT_AixConfig.Motor.SpeedSetpointWindow));
	    END_REGION

	END_REGION

	(* REGION 9 - Reading actual position

	    REGION 9.1 - Left Motor

	        #sx_LeftServoHomeHasBeenSet := #iUDT_AixInputsModule.ServoStatusLeft.%X1;
	        IF #ix_MotorPositionId = #ci_Left
	        THEN
	            IF #sx_LeftServoHomeHasBeenSet THEN
	                #si_LastLeftMotorPosition := 0;
	            END_IF;
	            // Add last position change to static memory
	            #si_LeftMotorPosition += - #si_LastLeftMotorPosition;
	            // Save last motor position
	            #si_LastLeftMotorPosition := #iUDT_AixInputsModule.ServoLocationLeft;

	            // Copy displacement if motor position change is greater or equal to 1 cm and store rest
	            IF #si_LeftMotorPosition > 10 THEN
	                #iqUDT_ConveyorInterface.DeltaPosition := REAL_TO_INT(INT_TO_REAL(#si_LeftMotorPosition) * #iUDT_AixConfig.Motor.Ratio) / 10;
	                #si_LeftMotorPosition := #si_LeftMotorPosition MOD 10;
	            ELSE
	                #iqUDT_ConveyorInterface.DeltaPosition := 0;
	            END_IF;

	            // allocate Motor Rotation status
	            #sb_MotorRotationStatus.%X0 := #iUDT_AixInputsModule.LeftMotorDiagnostic.MotorStatus1;
	            #sb_MotorRotationStatus.%X1 := #iUDT_AixInputsModule.LeftMotorDiagnostic.MotorStatus2;

	            // Change direction sign if motor running reverse
	            IF ((#sb_MotorRotationStatus = #cb_MotorInCW) AND NOT #iUDT_AixConfig.Motor.DirectionReversal) OR
	                ((#sb_MotorRotationStatus = #cb_MotorInCCW) AND #iUDT_AixConfig.Motor.DirectionReversal)
	            THEN

	                #iqUDT_ConveyorInterface.DeltaPosition *= -1;

	            END_IF;

	            // Motor positioned
	            #qx_Positioned := #iUDT_AixInputsModule.ServoStatusLeft.%X0;

	        END_IF;

	    END_REGION

	    REGION 9.2 - Right motor
	        #sx_RightServoHomeHasBeenSet := #iUDT_AixInputsModule.ServoStatusRight.%X1;
	        IF #ix_MotorPositionId = #ci_Right
	        THEN
	            IF #sx_RightServoHomeHasBeenSet THEN
	                #si_LastRightMotorPosition := 0;
	            END_IF;
	            // Add last position change to static memory
	            #si_RightMotorPosition += - #si_LastRightMotorPosition;
	            // Save last motor position
	            #si_LastRightMotorPosition := #iUDT_AixInputsModule.ServoLocationRight;

	            // Copy displacement if motor position change is greater or equal to 1 cm and store rest
	            IF #si_RightMotorPosition > 10 THEN
	                #iqUDT_ConveyorInterface.DeltaPosition := REAL_TO_INT(INT_TO_REAL(#si_RightMotorPosition) * #iUDT_AixConfig.Motor.Ratio) / 10;
	                #si_RightMotorPosition := #si_RightMotorPosition MOD 10;
	            ELSE
	                #iqUDT_ConveyorInterface.DeltaPosition := 0;
	            END_IF;

	            // allocate Motor Rotation status
	            #sb_MotorRotationStatus.%X0 := #iUDT_AixInputsModule.RightMotorDiagnostic.MotorStatus1;
	            #sb_MotorRotationStatus.%X1 := #iUDT_AixInputsModule.RightMotorDiagnostic.MotorStatus2;

	            // Change direction sign if motor running reverse
	            IF ((#sb_MotorRotationStatus = #cb_MotorInCW) AND NOT #iUDT_AixConfig.Motor.DirectionReversal) OR
	                ((#sb_MotorRotationStatus = #cb_MotorInCCW) AND #iUDT_AixConfig.Motor.DirectionReversal)
	            THEN

	                #iqUDT_ConveyorInterface.DeltaPosition *= -1;

	            END_IF;

	            // Motor positioned
	            #qx_Positioned := #iUDT_AixInputsModule.ServoStatusRight.%X0;

	        END_IF;

	    END_REGION


	END_REGION *)

	REGION 9 - Reading actual position

	    REGION 9.1 - Left motor

	        IF #ii_MotorPositionId = #ci_Master_Left OR #ii_MotorPositionId = #ci_Slave_Left
	        THEN
	            IF #iUDT_AixInputsModule.ServoLocationLeft = 0 THEN
	                #si_LastLeftMotorPosition := 0;
	            END_IF;
	            // Add last position change to static memory
	            #si_LeftMotorPosition += ABS(ABS(#iUDT_AixInputsModule.ServoLocationLeft) - ABS(#si_LastLeftMotorPosition));
	            // Save last motor position
	            #si_LastLeftMotorPosition := #iUDT_AixInputsModule.ServoLocationLeft;

	            // Copy delta position if motor position change is greater or equal to 1 cm and store rest
	            IF #si_LeftMotorPosition > 10 THEN
	                IF #ii_MotorPositionId = #ci_Master_Left THEN
	                    #iqUDT_ConveyorInterface.DeltaPosition := REAL_TO_INT(INT_TO_REAL(#si_LeftMotorPosition) * #iUDT_AixConfig.Motor.Ratio) / 10;
	                END_IF;
	                #si_LeftMotorPosition := #si_LeftMotorPosition MOD 10;
	            ELSE
	                IF #ii_MotorPositionId = #ci_Master_Left THEN
	                    #iqUDT_ConveyorInterface.DeltaPosition := 0;
	                END_IF;
	            END_IF;
	            // Change direction sign if motor running reverse
	            IF #iUDT_AixInputsModule.LeftMotorDiagnostic.MotorStatus1 AND NOT #iUDT_AixInputsModule.LeftMotorDiagnostic.MotorStatus2 AND NOT #iUDT_AixConfig.Motor.DirectionReversal
	                OR NOT #iUDT_AixInputsModule.LeftMotorDiagnostic.MotorStatus1 AND #iUDT_AixInputsModule.LeftMotorDiagnostic.MotorStatus2 AND #iUDT_AixConfig.Motor.DirectionReversal
	            THEN
	                IF #ii_MotorPositionId = #ci_Master_Left THEN
	                    #iqUDT_ConveyorInterface.DeltaPosition *= -1;
	                END_IF;
	            END_IF;

	            // Motor positioned
	            #qx_Positioned := #iUDT_AixInputsModule.ServoStatusLeft.%X0;

	        END_IF;

	    END_REGION

	    REGION 9.2 - Right motor

	        IF #ii_MotorPositionId = #ci_Master_Right OR #ii_MotorPositionId = #ci_Slave_Right
	        THEN
	            IF #iUDT_AixInputsModule.ServoLocationRight = 0 THEN
	                #si_LastRightMotorPosition := 0;
	            END_IF;
	            // Add last position change to static memory
	            #si_RightMotorPosition += ABS(ABS(#iUDT_AixInputsModule.ServoLocationRight) - ABS(#si_LastRightMotorPosition));
	            // Save last motor position
	            #si_LastRightMotorPosition := #iUDT_AixInputsModule.ServoLocationRight;

	            // Copy delta position if motor position change is greater or equal to 1 cm and store rest
	            IF #si_RightMotorPosition > 10 THEN
	                IF #ii_MotorPositionId = #ci_Master_Right THEN
	                    #iqUDT_ConveyorInterface.DeltaPosition := REAL_TO_INT(INT_TO_REAL(#si_RightMotorPosition) * #iUDT_AixConfig.Motor.Ratio) / 10;
	                END_IF;
	                #si_RightMotorPosition := #si_RightMotorPosition MOD 10;
	            ELSE
	                IF #ii_MotorPositionId = #ci_Master_Right THEN
	                    #iqUDT_ConveyorInterface.DeltaPosition := 0;
	                END_IF;
	            END_IF;
	            // Change direction sign if motor running reverse
	            IF #iUDT_AixInputsModule.RightMotorDiagnostic.MotorStatus1 AND NOT #iUDT_AixInputsModule.RightMotorDiagnostic.MotorStatus2 AND NOT #iUDT_AixConfig.Motor.DirectionReversal
	                OR NOT #iUDT_AixInputsModule.RightMotorDiagnostic.MotorStatus1 AND #iUDT_AixInputsModule.RightMotorDiagnostic.MotorStatus2 AND #iUDT_AixConfig.Motor.DirectionReversal
	            THEN
	                IF #ii_MotorPositionId = #ci_Master_Right THEN
	                    #iqUDT_ConveyorInterface.DeltaPosition *= -1;
	                END_IF;
	            END_IF;

	            // Motor positioned
	            #qx_Positioned := #iUDT_AixInputsModule.ServoStatusRight.%X0;

	        END_IF;

	    END_REGION

	END_REGION


	REGION 10 - Copy signals to interface DB and to status output UDT

	    REGION 10.1 - Motor

	        // Create internal error status
	        // Write Conveyor interface bits only if it is a Master
	        IF #ii_MotorPositionId = #ci_Master_Left OR #ii_MotorPositionId = #ci_Master_Right THEN

	            #iqUDT_ConveyorInterface.VFDRunning := #sx_AixAvailableControler AND
	            (#si_ActualSpeed <> 0);                 // Write true on output Conveyor interface structure if Ai2's are in operation and motor is turning

